LIN {X 0.171,Y -429.306,Z 1097.500,A 0.000,B 0.000,C 90.000,E1 269.943} C_DIS
LIN {X 0.033,Y -421.795,Z 1097.499,A 0.000,B 0.000,C 90.000,E1 269.771} C_DIS
LIN {X 0.153,Y -409.790,Z 1097.498,A 0.000,B 0.000,C 90.000,E1 269.542} C_DIS
LIN {X -0.190,Y -399.220,Z 1097.497,A 0.000,B 0.000,C 90.000,E1 269.484} C_DIS
LIN {X -0.102,Y -389.692,Z 1097.497,A 0.000,B 0.000,C 90.000,E1 269.427} C_DIS
LIN {X -0.076,Y -181.414,Z 1097.497,A 0.000,B 0.000,C 90.000,E1 269.427} C_DIS
LIN {X 0.018,Y -180.819,Z 1097.471,A 0.000,B 0.000,C 90.000,E1 264.837} C_DIS
LIN {X -0.083,Y -178.922,Z 1097.443,A 0.000,B 0.000,C 90.000,E1 259.803} C_DIS
LIN {X 0.003,Y -175.968,Z 1097.415,A 0.000,B 0.000,C 90.000,E1 254.685} C_DIS
LIN {X -0.050,Y -175.450,Z 1097.410,A 0.000,B 0.000,C 90.000,E1 253.850} C_DIS
LIN {X -0.041,Y -172.203,Z 1097.386,A 0.000,B 0.000,C 90.000,E1 249.571} C_DIS
LIN {X -0.062,Y -171.678,Z 1097.382,A 0.000,B 0.000,C 90.000,E1 248.720} C_DIS
LIN {X -0.072,Y -167.904,Z 1097.358,A 0.000,B 0.000,C 90.000,E1 244.409} C_DIS
LIN {X -0.053,Y -166.644,Z 1097.348,A 0.000,B 0.000,C 90.000,E1 242.666} C_DIS
LIN {X 0.002,Y -162.628,Z 1097.324,A 0.000,B 0.000,C 90.000,E1 238.280} C_DIS
LIN {X 0.061,Y -161.316,Z 1097.314,A 0.000,B 0.000,C 90.000,E1 236.501} C_DIS
LIN {X -0.029,Y -157.312,Z 1097.289,A 0.000,B 0.000,C 90.000,E1 232.110} C_DIS
LIN {X -0.097,Y -155.290,Z 1097.275,A 0.000,B 0.000,C 90.000,E1 229.461} C_DIS
LIN {X 0.050,Y -151.653,Z 1097.250,A 0.000,B 0.000,C 90.000,E1 224.919} C_DIS
LIN {X -0.013,Y -150.520,Z 1097.240,A 0.000,B 0.000,C 90.000,E1 223.137} C_DIS
LIN {X 0.011,Y -147.245,Z 1097.214,A 0.000,B 0.000,C 90.000,E1 218.588} C_DIS
LIN {X -0.025,Y -145.270,Z 1097.194,A 0.000,B 0.000,C 90.000,E1 214.945} C_DIS
LIN {X 0.009,Y -142.377,Z 1097.163,A 0.000,B 0.000,C 90.000,E1 209.411} C_DIS
LIN {X 0.059,Y -141.353,Z 1097.148,A 0.000,B 0.000,C 90.000,E1 206.616} C_DIS
LIN {X 0.042,Y -139.340,Z 1097.112,A 0.000,B 0.000,C 90.000,E1 200.120} C_DIS
LIN {X -0.039,Y -139.007,Z 1097.102,A 0.000,B 0.000,C 90.000,E1 198.290} C_DIS
LIN {X 0.048,Y -138.340,Z 1097.055,A 0.000,B 0.000,C 90.000,E1 189.849} C_DIS
LIN {X 0.071,Y -139.403,Z 1097.008,A 0.000,B 0.000,C 90.000,E1 181.432} C_DIS
LIN {X -0.015,Y -141.310,Z 1096.972,A 0.000,B 0.000,C 90.000,E1 174.951} C_DIS
LIN {X -0.058,Y -142.670,Z 1096.956,A 0.000,B 0.000,C 90.000,E1 172.186} C_DIS
LIN {X 0.064,Y -145.019,Z 1096.931,A 0.000,B 0.000,C 90.000,E1 167.521} C_DIS
LIN {X 0.021,Y -147.646,Z 1096.910,A 0.000,B 0.000,C 90.000,E1 163.866} C_DIS
LIN {X -0.043,Y -150.280,Z 1096.890,A 0.000,B 0.000,C 90.000,E1 160.242} C_DIS
LIN {X -0.030,Y -153.684,Z 1096.870,A 0.000,B 0.000,C 90.000,E1 156.613} C_DIS
LIN {X 0.025,Y -157.098,Z 1096.850,A 0.000,B 0.000,C 90.000,E1 152.999} C_DIS
LIN {X -0.037,Y -161.237,Z 1096.830,A 0.000,B 0.000,C 90.000,E1 149.459} C_DIS
LIN {X 0.048,Y -163.325,Z 1096.820,A 0.000,B 0.000,C 90.000,E1 147.661} C_DIS
LIN {X -0.081,Y -167.778,Z 1096.801,A 0.000,B 0.000,C 90.000,E1 144.196} C_DIS
LIN {X 0.071,Y -171.592,Z 1096.786,A 0.000,B 0.000,C 90.000,E1 141.537} C_DIS
LIN {X 0.002,Y -176.543,Z 1096.767,A 0.000,B 0.000,C 90.000,E1 138.119} C_DIS
LIN {X -0.006,Y -180.842,Z 1096.753,A 0.000,B 0.000,C 90.000,E1 135.567} C_DIS
LIN {X -0.022,Y -186.253,Z 1096.734,A 0.000,B 0.000,C 90.000,E1 132.204} C_DIS
LIN {X -0.084,Y -190.889,Z 1096.721,A 0.000,B 0.000,C 90.000,E1 129.725} C_DIS
LIN {X -0.051,Y -196.654,Z 1096.702,A 0.000,B 0.000,C 90.000,E1 126.423} C_DIS
LIN {X -0.056,Y -200.011,Z 1096.693,A 0.000,B 0.000,C 90.000,E1 124.739} C_DIS
LIN {X 0.114,Y -308.191,Z 1096.693,A 0.000,B 0.000,C 90.000,E1 124.692} C_DIS
LIN {X -0.031,Y -313.358,Z 1096.692,A 0.000,B 0.000,C 90.000,E1 124.532} C_DIS
LIN {X 0.081,Y -315.849,Z 1096.691,A 0.000,B 0.000,C 90.000,E1 124.326} C_DIS
LIN {X -0.136,Y -319.180,Z 1096.689,A 0.000,B 0.000,C 90.000,E1 123.992} C_DIS
LIN {X 0.031,Y -321.119,Z 1096.687,A 0.000,B 0.000,C 90.000,E1 123.658} C_DIS
LIN {X -0.070,Y -322.635,Z 1096.685,A 0.000,B 0.000,C 90.000,E1 123.372} C_DIS
LIN {X -0.076,Y -326.114,Z 1096.680,A 0.000,B 0.000,C 90.000,E1 122.418} C_DIS
LIN {X -0.078,Y -336.920,Z 1096.664,A 0.000,B 0.000,C 90.000,E1 119.589} C_DIS
LIN {X 0.023,Y -349.100,Z 1096.649,A 0.000,B 0.000,C 90.000,E1 116.796} C_DIS
LIN {X 0.009,Y -362.765,Z 1096.634,A 0.000,B 0.000,C 90.000,E1 114.079} C_DIS
LIN {X -0.006,Y -376.251,Z 1096.621,A 0.000,B 0.000,C 90.000,E1 111.716} C_DIS
LIN {X 0.043,Y -391.099,Z 1096.608,A 0.000,B 0.000,C 90.000,E1 109.396} C_DIS
LIN {X -0.045,Y -407.413,Z 1096.595,A 0.000,B 0.000,C 90.000,E1 107.149} C_DIS
LIN {X -0.100,Y -425.309,Z 1096.583,A 0.000,B 0.000,C 90.000,E1 104.954} C_DIS
LIN {X -0.142,Y -444.799,Z 1096.571,A 0.000,B 0.000,C 90.000,E1 102.827} C_DIS
LIN {X -0.016,Y -465.050,Z 1096.560,A 0.000,B 0.000,C 90.000,E1 100.838} C_DIS
LIN {X 0.001,Y -467.605,Z 1096.559,A 0.000,B 0.000,C 90.000,E1 100.602} C_DIS
LIN {X 0.018,Y -469.774,Z 1096.558,A 0.000,B 0.000,C 90.000,E1 100.366} C_DIS
LIN {X -0.217,Y -471.537,Z 1096.556,A 0.000,B 0.000,C 90.000,E1 100.141} C_DIS
LIN {X 0.098,Y -472.861,Z 1096.555,A 0.000,B 0.000,C 90.000,E1 99.849} C_DIS
LIN {X -0.186,Y -474.513,Z 1096.552,A 0.000,B 0.000,C 90.000,E1 99.378} C_DIS
LIN {X -0.072,Y -475.101,Z 1096.549,A 0.000,B 0.000,C 90.000,E1 98.859} C_DIS
LIN {X 0.056,Y -474.725,Z 1096.546,A 0.000,B 0.000,C 90.000,E1 98.341} C_DIS
LIN {X 0.253,Y -473.330,Z 1096.544,A 0.000,B 0.000,C 90.000,E1 97.814} C_DIS
LIN {X 0.050,Y -472.179,Z 1096.542,A 0.000,B 0.000,C 90.000,E1 97.587} C_DIS
LIN {X -0.088,Y -470.646,Z 1096.541,A 0.000,B 0.000,C 90.000,E1 97.352} C_DIS
LIN {X -0.214,Y -456.164,Z 1096.530,A 0.000,B 0.000,C 90.000,E1 95.334} C_DIS
LIN {X -0.079,Y -440.261,Z 1096.516,A 0.000,B 0.000,C 90.000,E1 92.980} C_DIS
LIN {X 0.048,Y -425.629,Z 1096.503,A 0.000,B 0.000,C 90.000,E1 90.573} C_DIS
LIN {X 0.049,Y -407.500,Z 1096.485,A 0.000,B 0.000,C 90.000,E1 87.306} C_DIS
LIN {X 0.079,Y -397.005,Z 1096.474,A 0.000,B 0.000,C 90.000,E1 85.355} C_DIS
LIN {X -0.034,Y -386.300,Z 1096.463,A 0.000,B 0.000,C 90.000,E1 83.394} C_DIS
LIN {X 0.053,Y -377.169,Z 1096.454,A 0.000,B 0.000,C 90.000,E1 81.659} C_DIS
LIN {X -0.034,Y -367.668,Z 1096.444,A 0.000,B 0.000,C 90.000,E1 79.926} C_DIS
LIN {X -0.166,Y -357.876,Z 1096.434,A 0.000,B 0.000,C 90.000,E1 78.173} C_DIS
LIN {X -0.039,Y -346.268,Z 1096.422,A 0.000,B 0.000,C 90.000,E1 76.047} C_DIS
LIN {X 0.148,Y -333.118,Z 1096.409,A 0.000,B 0.000,C 90.000,E1 73.559} C_DIS
LIN {X 0.013,Y -315.862,Z 1096.390,A 0.000,B 0.000,C 90.000,E1 70.115} C_DIS
LIN {X -0.145,Y -302.718,Z 1096.373,A 0.000,B 0.000,C 90.000,E1 67.230} C_DIS
LIN {X -0.035,Y -292.864,Z 1096.360,A 0.000,B 0.000,C 90.000,E1 64.897} C_DIS
LIN {X -0.178,Y -281.874,Z 1096.346,A 0.000,B 0.000,C 90.000,E1 62.231} C_DIS
LIN {X -0.070,Y -271.125,Z 1096.330,A 0.000,B 0.000,C 90.000,E1 59.459} C_DIS
LIN {X -0.053,Y -259.422,Z 1096.313,A 0.000,B 0.000,C 90.000,E1 56.294} C_DIS
LIN {X 0.000,Y -248.215,Z 1096.295,A 0.000,B 0.000,C 90.000,E1 53.050} C_DIS
LIN {X -0.007,Y -237.844,Z 1096.276,A 0.000,B 0.000,C 90.000,E1 49.747} C_DIS
LIN {X -0.005,Y -228.242,Z 1096.258,A 0.000,B 0.000,C 90.000,E1 46.377} C_DIS
LIN {X -0.035,Y -220.174,Z 1096.241,A 0.000,B 0.000,C 90.000,E1 43.338} C_DIS
LIN {X -0.086,Y -212.478,Z 1096.224,A 0.000,B 0.000,C 90.000,E1 40.253} C_DIS
LIN {X 0.013,Y -205.151,Z 1096.206,A 0.000,B 0.000,C 90.000,E1 37.076} C_DIS
LIN {X 0.052,Y -198.373,Z 1096.188,A 0.000,B 0.000,C 90.000,E1 33.865} C_DIS
LIN {X -0.122,Y -192.214,Z 1096.170,A 0.000,B 0.000,C 90.000,E1 30.669} C_DIS
LIN {X 0.023,Y -186.724,Z 1096.152,A 0.000,B 0.000,C 90.000,E1 27.334} C_DIS
LIN {X -0.055,Y -181.962,Z 1096.133,A 0.000,B 0.000,C 90.000,E1 24.027} C_DIS
LIN {X -0.053,Y -176.995,Z 1096.110,A 0.000,B 0.000,C 90.000,E1 19.812} C_DIS
LIN {X -0.055,Y -173.062,Z 1096.086,A 0.000,B 0.000,C 90.000,E1 15.552} C_DIS
LIN {X 0.016,Y -169.745,Z 1096.058,A 0.000,B 0.000,C 90.000,E1 10.366} C_DIS
LIN {X -0.011,Y -167.547,Z 1096.019,A 0.000,B 0.000,C 90.000,E1 3.440} C_DIS
LIN {X -0.017,Y -168.706,Z 1095.964,A 0.000,B 0.000,C 90.000,E1 353.451} C_DIS
LIN {X 0.055,Y -171.259,Z 1095.935,A 0.000,B 0.000,C 90.000,E1 348.229} C_DIS
LIN {X 0.070,Y -174.548,Z 1095.911,A 0.000,B 0.000,C 90.000,E1 343.921} C_DIS
LIN {X -0.075,Y -178.893,Z 1095.887,A 0.000,B 0.000,C 90.000,E1 339.699} C_DIS
LIN {X -0.044,Y -183.100,Z 1095.868,A 0.000,B 0.000,C 90.000,E1 336.305} C_DIS
LIN {X -0.023,Y -188.059,Z 1095.850,A 0.000,B 0.000,C 90.000,E1 332.948} C_DIS
LIN {X 0.046,Y -193.760,Z 1095.831,A 0.000,B 0.000,C 90.000,E1 329.616} C_DIS
LIN {X -0.047,Y -200.207,Z 1095.813,A 0.000,B 0.000,C 90.000,E1 326.373} C_DIS
LIN {X 0.027,Y -207.316,Z 1095.795,A 0.000,B 0.000,C 90.000,E1 323.130} C_DIS
LIN {X -0.076,Y -215.345,Z 1095.778,A 0.000,B 0.000,C 90.000,E1 319.989} C_DIS
LIN {X -0.018,Y -224.059,Z 1095.760,A 0.000,B 0.000,C 90.000,E1 316.863} C_DIS
LIN {X 0.089,Y -233.756,Z 1095.743,A 0.000,B 0.000,C 90.000,E1 313.785} C_DIS
LIN {X -0.018,Y -243.414,Z 1095.729,A 0.000,B 0.000,C 90.000,E1 311.191} C_DIS
LIN {X -0.037,Y -252.645,Z 1095.717,A 0.000,B 0.000,C 90.000,E1 308.991} C_DIS
LIN {X 0.077,Y -266.395,Z 1095.701,A 0.000,B 0.000,C 90.000,E1 306.091} C_DIS
LIN {X 0.080,Y -281.412,Z 1095.685,A 0.000,B 0.000,C 90.000,E1 303.293} C_DIS
LIN {X -0.005,Y -299.593,Z 1095.668,A 0.000,B 0.000,C 90.000,E1 300.256} C_DIS
LIN {X -0.016,Y -319.577,Z 1095.652,A 0.000,B 0.000,C 90.000,E1 297.308} C_DIS
LIN {X 0.009,Y -336.467,Z 1095.639,A 0.000,B 0.000,C 90.000,E1 295.079} C_DIS
LIN {X -0.080,Y -349.541,Z 1095.631,A 0.000,B 0.000,C 90.000,E1 293.567} C_DIS
LIN {X -0.194,Y -362.823,Z 1095.623,A 0.000,B 0.000,C 90.000,E1 292.153} C_DIS
LIN {X -0.066,Y -376.176,Z 1095.616,A 0.000,B 0.000,C 90.000,E1 290.844} C_DIS
LIN {X -0.076,Y -395.554,Z 1095.606,A 0.000,B 0.000,C 90.000,E1 289.141} C_DIS
LIN {X 0.030,Y -409.102,Z 1095.600,A 0.000,B 0.000,C 90.000,E1 287.946} C_DIS
LIN {X 0.036,Y -419.690,Z 1095.594,A 0.000,B 0.000,C 90.000,E1 286.985} C_DIS
LIN {X -0.079,Y -427.432,Z 1095.590,A 0.000,B 0.000,C 90.000,E1 286.260} C_DIS
LIN {X 0.023,Y -434.966,Z 1095.586,A 0.000,B 0.000,C 90.000,E1 285.481} C_DIS
LIN {X -0.185,Y -442.194,Z 1095.582,A 0.000,B 0.000,C 90.000,E1 284.717} C_DIS
LIN {X 0.151,Y -448.956,Z 1095.577,A 0.000,B 0.000,C 90.000,E1 283.883} C_DIS
LIN {X -0.002,Y -455.110,Z 1095.573,A 0.000,B 0.000,C 90.000,E1 283.119} C_DIS
LIN {X 0.075,Y -458.896,Z 1095.570,A 0.000,B 0.000,C 90.000,E1 282.591} C_DIS
LIN {X 0.013,Y -463.916,Z 1095.566,A 0.000,B 0.000,C 90.000,E1 281.827} C_DIS
LIN {X -0.104,Y -468.213,Z 1095.561,A 0.000,B 0.000,C 90.000,E1 281.074} C_DIS
LIN {X -0.089,Y -471.792,Z 1095.557,A 0.000,B 0.000,C 90.000,E1 280.310} C_DIS
LIN {X -0.130,Y -474.745,Z 1095.553,A 0.000,B 0.000,C 90.000,E1 279.557} C_DIS
LIN {X 0.060,Y -476.344,Z 1095.550,A 0.000,B 0.000,C 90.000,E1 279.029} C_DIS
LIN {X 0.187,Y -477.748,Z 1095.547,A 0.000,B 0.000,C 90.000,E1 278.511} C_DIS
LIN {X -0.147,Y -478.896,Z 1095.545,A 0.000,B 0.000,C 90.000,E1 278.049} C_DIS
LIN {X 0.002,Y -479.796,Z 1095.542,A 0.000,B 0.000,C 90.000,E1 277.530} C_DIS
LIN {X 0.159,Y -480.516,Z 1095.539,A 0.000,B 0.000,C 90.000,E1 277.011} C_DIS
LIN {X -0.100,Y -480.986,Z 1095.536,A 0.000,B 0.000,C 90.000,E1 276.543} C_DIS
LIN {X 0.013,Y -481.163,Z 1095.534,A 0.000,B 0.000,C 90.000,E1 276.030} C_DIS
LIN {X 0.183,Y -480.992,Z 1095.531,A 0.000,B 0.000,C 90.000,E1 275.511} C_DIS
LIN {X -0.127,Y -480.502,Z 1095.528,A 0.000,B 0.000,C 90.000,E1 275.049} C_DIS
LIN {X 0.040,Y -479.609,Z 1095.525,A 0.000,B 0.000,C 90.000,E1 274.531} C_DIS
LIN {X 0.200,Y -478.204,Z 1095.522,A 0.000,B 0.000,C 90.000,E1 274.012} C_DIS
LIN {X -0.153,Y -476.301,Z 1095.520,A 0.000,B 0.000,C 90.000,E1 273.555} C_DIS
LIN {X -0.009,Y -473.740,Z 1095.517,A 0.000,B 0.000,C 90.000,E1 273.037} C_DIS
LIN {X 0.092,Y -470.356,Z 1095.514,A 0.000,B 0.000,C 90.000,E1 272.522} C_DIS
LIN {X 0.176,Y -466.075,Z 1095.511,A 0.000,B 0.000,C 90.000,E1 272.007} C_DIS
LIN {X -0.209,Y -460.563,Z 1095.508,A 0.000,B 0.000,C 90.000,E1 271.547} C_DIS
LIN {X -0.209,Y -457.683,Z 1095.507,A 0.000,B 0.000,C 90.000,E1 271.318} C_DIS
LIN {X 0.070,Y -451.340,Z 1095.505,A 0.000,B 0.000,C 90.000,E1 270.859} C_DIS
LIN {X -0.058,Y -444.673,Z 1095.503,A 0.000,B 0.000,C 90.000,E1 270.516} C_DIS
LIN {X -0.168,Y -437.586,Z 1095.501,A 0.000,B 0.000,C 90.000,E1 270.229} C_DIS
LIN {X 0.135,Y -430.141,Z 1095.500,A 0.000,B 0.000,C 90.000,E1 269.943} C_DIS
LIN {X -0.039,Y -422.384,Z 1095.499,A 0.000,B 0.000,C 90.000,E1 269.771} C_DIS
LIN {X 0.123,Y -414.688,Z 1095.498,A 0.000,B 0.000,C 90.000,E1 269.599} C_DIS
LIN {X 0.116,Y -406.084,Z 1095.497,A 0.000,B 0.000,C 90.000,E1 269.484} C_DIS
LIN {X -0.095,Y -394.535,Z 1095.497,A 0.000,B 0.000,C 90.000,E1 269.427} C_DIS
LIN {X -0.159,Y -391.661,Z 1095.497,A 0.000,B 0.000,C 90.000,E1 269.427} C_DIS
LIN {X 0.078,Y -181.412,Z 1095.497,A 0.000,B 0.000,C 90.000,E1 269.370} C_DIS
LIN {X -0.012,Y -180.816,Z 1095.471,A 0.000,B 0.000,C 90.000,E1 264.837} C_DIS
LIN {X 0.066,Y -178.919,Z 1095.443,A 0.000,B 0.000,C 90.000,E1 259.746} C_DIS
LIN {X -0.025,Y -175.964,Z 1095.415,A 0.000,B 0.000,C 90.000,E1 254.685} C_DIS
LIN {X 0.090,Y -175.441,Z 1095.410,A 0.000,B 0.000,C 90.000,E1 253.795} C_DIS
LIN {X -0.068,Y -172.198,Z 1095.386,A 0.000,B 0.000,C 90.000,E1 249.571} C_DIS
LIN {X -0.091,Y -171.671,Z 1095.382,A 0.000,B 0.000,C 90.000,E1 248.720} C_DIS
LIN {X -0.099,Y -167.897,Z 1095.358,A 0.000,B 0.000,C 90.000,E1 244.409} C_DIS
LIN {X 0.068,Y -166.636,Z 1095.348,A 0.000,B 0.000,C 90.000,E1 242.615} C_DIS
LIN {X -0.025,Y -162.622,Z 1095.324,A 0.000,B 0.000,C 90.000,E1 238.280} C_DIS
LIN {X 0.034,Y -161.308,Z 1095.314,A 0.000,B 0.000,C 90.000,E1 236.501} C_DIS
LIN {X -0.056,Y -157.305,Z 1095.289,A 0.000,B 0.000,C 90.000,E1 232.110} C_DIS
LIN {X 0.096,Y -155.281,Z 1095.275,A 0.000,B 0.000,C 90.000,E1 229.380} C_DIS
LIN {X 0.024,Y -151.646,Z 1095.250,A 0.000,B 0.000,C 90.000,E1 224.919} C_DIS
LIN {X -0.039,Y -150.515,Z 1095.240,A 0.000,B 0.000,C 90.000,E1 223.137} C_DIS
LIN {X -0.015,Y -147.239,Z 1095.214,A 0.000,B 0.000,C 90.000,E1 218.588} C_DIS
LIN {X -0.050,Y -145.263,Z 1095.194,A 0.000,B 0.000,C 90.000,E1 214.945} C_DIS
LIN {X -0.016,Y -142.373,Z 1095.163,A 0.000,B 0.000,C 90.000,E1 209.411} C_DIS
LIN {X -0.020,Y -141.758,Z 1095.153,A 0.000,B 0.000,C 90.000,E1 207.564} C_DIS
LIN {X 0.030,Y -139.498,Z 1095.117,A 0.000,B 0.000,C 90.000,E1 201.046} C_DIS
LIN {X 0.067,Y -139.004,Z 1095.101,A 0.000,B 0.000,C 90.000,E1 198.236} C_DIS
LIN {X 0.024,Y -138.339,Z 1095.055,A 0.000,B 0.000,C 90.000,E1 189.849} C_DIS
LIN {X 0.046,Y -139.406,Z 1095.008,A 0.000,B 0.000,C 90.000,E1 181.432} C_DIS
LIN {X -0.040,Y -141.314,Z 1094.972,A 0.000,B 0.000,C 90.000,E1 174.951} C_DIS
LIN {X 0.057,Y -142.673,Z 1094.956,A 0.000,B 0.000,C 90.000,E1 172.129} C_DIS
LIN {X 0.039,Y -145.026,Z 1094.931,A 0.000,B 0.000,C 90.000,E1 167.521} C_DIS
LIN {X -0.005,Y -147.652,Z 1094.910,A 0.000,B 0.000,C 90.000,E1 163.866} C_DIS
LIN {X -0.070,Y -150.288,Z 1094.890,A 0.000,B 0.000,C 90.000,E1 160.242} C_DIS
LIN {X -0.057,Y -153.695,Z 1094.870,A 0.000,B 0.000,C 90.000,E1 156.613} C_DIS
LIN {X -0.002,Y -157.108,Z 1094.850,A 0.000,B 0.000,C 90.000,E1 152.999} C_DIS
LIN {X -0.065,Y -161.250,Z 1094.830,A 0.000,B 0.000,C 90.000,E1 149.459} C_DIS
LIN {X 0.021,Y -163.336,Z 1094.820,A 0.000,B 0.000,C 90.000,E1 147.661} C_DIS
LIN {X 0.027,Y -167.791,Z 1094.801,A 0.000,B 0.000,C 90.000,E1 144.149} C_DIS
LIN {X 0.043,Y -171.605,Z 1094.786,A 0.000,B 0.000,C 90.000,E1 141.537} C_DIS
LIN {X 0.091,Y -176.559,Z 1094.767,A 0.000,B 0.000,C 90.000,E1 138.081} C_DIS
LIN {X -0.036,Y -180.857,Z 1094.753,A 0.000,B 0.000,C 90.000,E1 135.567} C_DIS
LIN {X -0.051,Y -186.269,Z 1094.734,A 0.000,B 0.000,C 90.000,E1 132.204} C_DIS
LIN {X 0.008,Y -190.905,Z 1094.720,A 0.000,B 0.000,C 90.000,E1 129.688} C_DIS
LIN {X 0.076,Y -196.671,Z 1094.702,A 0.000,B 0.000,C 90.000,E1 126.377} C_DIS
LIN {X 0.062,Y -199.941,Z 1094.693,A 0.000,B 0.000,C 90.000,E1 124.739} C_DIS
LIN {X 0.059,Y -307.476,Z 1094.693,A 0.000,B 0.000,C 90.000,E1 124.739} C_DIS
LIN {X 0.066,Y -309.988,Z 1094.693,A 0.000,B 0.000,C 90.000,E1 124.692} C_DIS
LIN {X -0.080,Y -313.832,Z 1094.692,A 0.000,B 0.000,C 90.000,E1 124.532} C_DIS
LIN {X 0.032,Y -316.142,Z 1094.691,A 0.000,B 0.000,C 90.000,E1 124.326} C_DIS
LIN {X -0.185,Y -319.328,Z 1094.689,A 0.000,B 0.000,C 90.000,E1 123.992} C_DIS
LIN {X -0.074,Y -321.258,Z 1094.687,A 0.000,B 0.000,C 90.000,E1 123.658} C_DIS
LIN {X 0.217,Y -322.762,Z 1094.685,A 0.000,B 0.000,C 90.000,E1 123.293} C_DIS
LIN {X 0.051,Y -337.012,Z 1094.664,A 0.000,B 0.000,C 90.000,E1 119.539} C_DIS
LIN {X 0.168,Y -349.206,Z 1094.649,A 0.000,B 0.000,C 90.000,E1 116.744} C_DIS
LIN {X -0.161,Y -362.886,Z 1094.634,A 0.000,B 0.000,C 90.000,E1 114.079} C_DIS
LIN {X -0.180,Y -376.387,Z 1094.620,A 0.000,B 0.000,C 90.000,E1 111.716} C_DIS
LIN {X -0.134,Y -391.250,Z 1094.608,A 0.000,B 0.000,C 90.000,E1 109.396} C_DIS
LIN {X 0.164,Y -407.581,Z 1094.595,A 0.000,B 0.000,C 90.000,E1 107.094} C_DIS
LIN {X 0.127,Y -425.496,Z 1094.583,A 0.000,B 0.000,C 90.000,E1 104.898} C_DIS
LIN {X 0.109,Y -444.998,Z 1094.571,A 0.000,B 0.000,C 90.000,E1 102.771} C_DIS
LIN {X -0.192,Y -465.257,Z 1094.560,A 0.000,B 0.000,C 90.000,E1 100.838} C_DIS
LIN {X -0.174,Y -467.803,Z 1094.559,A 0.000,B 0.000,C 90.000,E1 100.602} C_DIS
LIN {X -0.157,Y -469.911,Z 1094.557,A 0.000,B 0.000,C 90.000,E1 100.366} C_DIS
LIN {X 0.155,Y -471.631,Z 1094.556,A 0.000,B 0.000,C 90.000,E1 100.074} C_DIS
LIN {X -0.077,Y -472.922,Z 1094.555,A 0.000,B 0.000,C 90.000,E1 99.849} C_DIS
LIN {X 0.107,Y -474.525,Z 1094.552,A 0.000,B 0.000,C 90.000,E1 99.321} C_DIS
LIN {X 0.224,Y -475.071,Z 1094.549,A 0.000,B 0.000,C 90.000,E1 98.803} C_DIS
LIN {X -0.118,Y -474.653,Z 1094.546,A 0.000,B 0.000,C 90.000,E1 98.341} C_DIS
LIN {X 0.079,Y -473.211,Z 1094.543,A 0.000,B 0.000,C 90.000,E1 97.814} C_DIS
LIN {X -0.123,Y -472.031,Z 1094.542,A 0.000,B 0.000,C 90.000,E1 97.587} C_DIS
LIN {X 0.206,Y -470.462,Z 1094.541,A 0.000,B 0.000,C 90.000,E1 97.296} C_DIS
LIN {X 0.069,Y -456.006,Z 1094.529,A 0.000,B 0.000,C 90.000,E1 95.277} C_DIS
LIN {X 0.191,Y -440.105,Z 1094.516,A 0.000,B 0.000,C 90.000,E1 92.922} C_DIS
LIN {X -0.121,Y -425.471,Z 1094.503,A 0.000,B 0.000,C 90.000,E1 90.573} C_DIS
LIN {X -0.118,Y -407.373,Z 1094.485,A 0.000,B 0.000,C 90.000,E1 87.306} C_DIS
LIN {X -0.086,Y -396.877,Z 1094.474,A 0.000,B 0.000,C 90.000,E1 85.355} C_DIS
LIN {X 0.187,Y -386.154,Z 1094.463,A 0.000,B 0.000,C 90.000,E1 83.337} C_DIS
LIN {X -0.108,Y -377.019,Z 1094.454,A 0.000,B 0.000,C 90.000,E1 81.659} C_DIS
LIN {X -0.129,Y -367.483,Z 1094.444,A 0.000,B 0.000,C 90.000,E1 79.916} C_DIS
LIN {X 0.024,Y -357.661,Z 1094.434,A 0.000,B 0.000,C 90.000,E1 78.117} C_DIS
LIN {X 0.138,Y -346.059,Z 1094.422,A 0.000,B 0.000,C 90.000,E1 75.992} C_DIS
LIN {X -0.124,Y -331.289,Z 1094.407,A 0.000,B 0.000,C 90.000,E1 73.268} C_DIS
LIN {X 0.153,Y -315.668,Z 1094.389,A 0.000,B 0.000,C 90.000,E1 70.061} C_DIS
LIN {X -0.021,Y -302.546,Z 1094.373,A 0.000,B 0.000,C 90.000,E1 67.177} C_DIS
LIN {X 0.077,Y -292.684,Z 1094.360,A 0.000,B 0.000,C 90.000,E1 64.845} C_DIS
LIN {X 0.051,Y -281.675,Z 1094.345,A 0.000,B 0.000,C 90.000,E1 62.153} C_DIS
LIN {X 0.012,Y -270.918,Z 1094.330,A 0.000,B 0.000,C 90.000,E1 59.410} C_DIS
LIN {X -0.105,Y -260.470,Z 1094.314,A 0.000,B 0.000,C 90.000,E1 56.628} C_DIS
LIN {X -0.040,Y -250.420,Z 1094.299,A 0.000,B 0.000,C 90.000,E1 53.749} C_DIS
LIN {X 0.055,Y -239.828,Z 1094.280,A 0.000,B 0.000,C 90.000,E1 50.436} C_DIS
LIN {X 0.100,Y -230.051,Z 1094.262,A 0.000,B 0.000,C 90.000,E1 47.067} C_DIS
LIN {X 0.111,Y -221.895,Z 1094.245,A 0.000,B 0.000,C 90.000,E1 44.028} C_DIS
LIN {X -0.068,Y -214.054,Z 1094.228,A 0.000,B 0.000,C 90.000,E1 40.987} C_DIS
LIN {X 0.070,Y -206.616,Z 1094.210,A 0.000,B 0.000,C 90.000,E1 37.810} C_DIS
LIN {X 0.095,Y -199.664,Z 1094.192,A 0.000,B 0.000,C 90.000,E1 34.612} C_DIS
LIN {X 0.051,Y -193.336,Z 1094.174,A 0.000,B 0.000,C 90.000,E1 31.386} C_DIS
LIN {X 0.049,Y -187.706,Z 1094.156,A 0.000,B 0.000,C 90.000,E1 28.103} C_DIS
LIN {X 0.070,Y -182.784,Z 1094.138,A 0.000,B 0.000,C 90.000,E1 24.771} C_DIS
LIN {X 0.074,Y -178.580,Z 1094.119,A 0.000,B 0.000,C 90.000,E1 21.408} C_DIS
LIN {X 0.058,Y -174.217,Z 1094.095,A 0.000,B 0.000,C 90.000,E1 17.166} C_DIS
LIN {X 0.044,Y -170.975,Z 1094.072,A 0.000,B 0.000,C 90.000,E1 12.883} C_DIS
LIN {X 0.035,Y -168.371,Z 1094.043,A 0.000,B 0.000,C 90.000,E1 7.701} C_DIS
LIN {X -0.056,Y -169.131,Z 1093.954,A 0.000,B 0.000,C 90.000,E1 351.724} C_DIS
LIN {X -0.015,Y -172.198,Z 1093.925,A 0.000,B 0.000,C 90.000,E1 346.520} C_DIS
LIN {X -0.045,Y -175.946,Z 1093.901,A 0.000,B 0.000,C 90.000,E1 342.236} C_DIS
LIN {X -0.039,Y -179.662,Z 1093.882,A 0.000,B 0.000,C 90.000,E1 338.827} C_DIS
LIN {X 0.013,Y -184.054,Z 1093.864,A 0.000,B 0.000,C 90.000,E1 335.433} C_DIS
LIN {X -0.029,Y -189.201,Z 1093.845,A 0.000,B 0.000,C 90.000,E1 332.103} C_DIS
LIN {X 0.000,Y -195.124,Z 1093.827,A 0.000,B 0.000,C 90.000,E1 328.791} C_DIS
LIN {X 0.057,Y -201.693,Z 1093.808,A 0.000,B 0.000,C 90.000,E1 325.515} C_DIS
LIN {X 0.013,Y -209.099,Z 1093.791,A 0.000,B 0.000,C 90.000,E1 322.316} C_DIS
LIN {X 0.018,Y -218.349,Z 1093.771,A 0.000,B 0.000,C 90.000,E1 318.771} C_DIS
LIN {X -0.011,Y -227.406,Z 1093.754,A 0.000,B 0.000,C 90.000,E1 315.688} C_DIS
LIN {X 0.066,Y -236.239,Z 1093.739,A 0.000,B 0.000,C 90.000,E1 313.014} C_DIS
LIN {X 0.041,Y -246.256,Z 1093.725,A 0.000,B 0.000,C 90.000,E1 310.415} C_DIS
LIN {X 0.050,Y -255.841,Z 1093.712,A 0.000,B 0.000,C 90.000,E1 308.222} C_DIS
LIN {X -0.072,Y -269.957,Z 1093.697,A 0.000,B 0.000,C 90.000,E1 305.391} C_DIS
LIN {X -0.140,Y -285.314,Z 1093.681,A 0.000,B 0.000,C 90.000,E1 302.625} C_DIS
LIN {X 0.142,Y -303.898,Z 1093.664,A 0.000,B 0.000,C 90.000,E1 299.539} C_DIS
LIN {X 0.124,Y -324.303,Z 1093.648,A 0.000,B 0.000,C 90.000,E1 296.616} C_DIS
LIN {X -0.159,Y -339.087,Z 1093.637,A 0.000,B 0.000,C 90.000,E1 294.771} C_DIS
LIN {X 0.076,Y -360.518,Z 1093.624,A 0.000,B 0.000,C 90.000,E1 292.333} C_DIS
LIN {X -0.095,Y -373.945,Z 1093.617,A 0.000,B 0.000,C 90.000,E1 291.046} C_DIS
LIN {X 0.129,Y -395.786,Z 1093.606,A 0.000,B 0.000,C 90.000,E1 289.087} C_DIS
LIN {X -0.193,Y -409.399,Z 1093.599,A 0.000,B 0.000,C 90.000,E1 287.946} C_DIS
LIN {X -0.144,Y -417.381,Z 1093.596,A 0.000,B 0.000,C 90.000,E1 287.221} C_DIS
LIN {X 0.183,Y -425.193,Z 1093.591,A 0.000,B 0.000,C 90.000,E1 286.441} C_DIS
LIN {X 0.003,Y -432.714,Z 1093.587,A 0.000,B 0.000,C 90.000,E1 285.717} C_DIS
LIN {X -0.173,Y -440.085,Z 1093.583,A 0.000,B 0.000,C 90.000,E1 284.954} C_DIS
LIN {X 0.145,Y -447.039,Z 1093.578,A 0.000,B 0.000,C 90.000,E1 284.120} C_DIS
LIN {X -0.020,Y -453.381,Z 1093.574,A 0.000,B 0.000,C 90.000,E1 283.355} C_DIS
LIN {X -0.136,Y -459.152,Z 1093.570,A 0.000,B 0.000,C 90.000,E1 282.591} C_DIS
LIN {X -0.198,Y -464.157,Z 1093.566,A 0.000,B 0.000,C 90.000,E1 281.827} C_DIS
LIN {X -0.066,Y -467.109,Z 1093.563,A 0.000,B 0.000,C 90.000,E1 281.299} C_DIS
LIN {X -0.154,Y -470.891,Z 1093.558,A 0.000,B 0.000,C 90.000,E1 280.546} C_DIS
LIN {X 0.020,Y -473.072,Z 1093.556,A 0.000,B 0.000,C 90.000,E1 280.018} C_DIS
LIN {X 0.128,Y -474.972,Z 1093.553,A 0.000,B 0.000,C 90.000,E1 279.500} C_DIS
LIN {X -0.149,Y -476.549,Z 1093.550,A 0.000,B 0.000,C 90.000,E1 279.029} C_DIS
LIN {X -0.022,Y -477.923,Z 1093.547,A 0.000,B 0.000,C 90.000,E1 278.511} C_DIS
LIN {X 0.119,Y -479.055,Z 1093.544,A 0.000,B 0.000,C 90.000,E1 277.992} C_DIS
LIN {X -0.206,Y -480.000,Z 1093.542,A 0.000,B 0.000,C 90.000,E1 277.530} C_DIS
LIN {X 0.011,Y -480.733,Z 1093.539,A 0.000,B 0.000,C 90.000,E1 277.004} C_DIS
LIN {X 0.171,Y -481.182,Z 1093.536,A 0.000,B 0.000,C 90.000,E1 276.486} C_DIS
LIN {X -0.141,Y -481.381,Z 1093.533,A 0.000,B 0.000,C 90.000,E1 276.024} C_DIS
LIN {X -0.021,Y -481.254,Z 1093.531,A 0.000,B 0.000,C 90.000,E1 275.511} C_DIS
LIN {X 0.151,Y -480.758,Z 1093.528,A 0.000,B 0.000,C 90.000,E1 274.992} C_DIS
LIN {X -0.160,Y -479.832,Z 1093.525,A 0.000,B 0.000,C 90.000,E1 274.531} C_DIS
LIN {X 0.002,Y -478.483,Z 1093.522,A 0.000,B 0.000,C 90.000,E1 274.012} C_DIS
LIN {X 0.127,Y -476.549,Z 1093.520,A 0.000,B 0.000,C 90.000,E1 273.498} C_DIS
LIN {X -0.202,Y -473.979,Z 1093.517,A 0.000,B 0.000,C 90.000,E1 273.037} C_DIS
LIN {X -0.099,Y -470.584,Z 1093.514,A 0.000,B 0.000,C 90.000,E1 272.522} C_DIS
LIN {X -0.012,Y -466.238,Z 1093.511,A 0.000,B 0.000,C 90.000,E1 272.007} C_DIS
LIN {X 0.067,Y -460.767,Z 1093.508,A 0.000,B 0.000,C 90.000,E1 271.489} C_DIS
LIN {X 0.021,Y -454.507,Z 1093.506,A 0.000,B 0.000,C 90.000,E1 271.031} C_DIS
LIN {X 0.058,Y -447.822,Z 1093.504,A 0.000,B 0.000,C 90.000,E1 270.630} C_DIS
LIN {X 0.159,Y -440.898,Z 1093.502,A 0.000,B 0.000,C 90.000,E1 270.286} C_DIS
LIN {X -0.153,Y -433.585,Z 1093.500,A 0.000,B 0.000,C 90.000,E1 270.057} C_DIS
LIN {X -0.034,Y -425.904,Z 1093.499,A 0.000,B 0.000,C 90.000,E1 269.828} C_DIS
LIN {X 0.035,Y -418.330,Z 1093.498,A 0.000,B 0.000,C 90.000,E1 269.656} C_DIS
LIN {X -0.080,Y -410.064,Z 1093.497,A 0.000,B 0.000,C 90.000,E1 269.542} C_DIS
LIN {X -0.086,Y -397.424,Z 1093.497,A 0.000,B 0.000,C 90.000,E1 269.427} C_DIS
LIN {X 0.120,Y -390.627,Z 1093.497,A 0.000,B 0.000,C 90.000,E1 269.370} C_DIS
LIN {X 0.027,Y -181.408,Z 1093.497,A 0.000,B 0.000,C 90.000,E1 269.370} C_DIS
LIN {X -0.061,Y -180.810,Z 1093.471,A 0.000,B 0.000,C 90.000,E1 264.837} C_DIS
LIN {X 0.016,Y -178.913,Z 1093.443,A 0.000,B 0.000,C 90.000,E1 259.746} C_DIS
LIN {X 0.095,Y -175.957,Z 1093.415,A 0.000,B 0.000,C 90.000,E1 254.629} C_DIS
LIN {X 0.042,Y -175.428,Z 1093.410,A 0.000,B 0.000,C 90.000,E1 253.795} C_DIS
LIN {X 0.045,Y -172.188,Z 1093.386,A 0.000,B 0.000,C 90.000,E1 249.518} C_DIS
LIN {X 0.021,Y -171.660,Z 1093.381,A 0.000,B 0.000,C 90.000,E1 248.666} C_DIS
LIN {X 0.005,Y -167.884,Z 1093.358,A 0.000,B 0.000,C 90.000,E1 244.357} C_DIS
LIN {X 0.020,Y -166.621,Z 1093.348,A 0.000,B 0.000,C 90.000,E1 242.615} C_DIS
LIN {X 0.014,Y -162.608,Z 1093.324,A 0.000,B 0.000,C 90.000,E1 238.250} C_DIS
LIN {X -0.013,Y -161.293,Z 1093.314,A 0.000,B 0.000,C 90.000,E1 236.501} C_DIS
LIN {X 0.022,Y -157.291,Z 1093.289,A 0.000,B 0.000,C 90.000,E1 232.065} C_DIS
LIN {X 0.045,Y -156.008,Z 1093.279,A 0.000,B 0.000,C 90.000,E1 230.275} C_DIS
LIN {X 0.005,Y -152.267,Z 1093.255,A 0.000,B 0.000,C 90.000,E1 225.810} C_DIS
LIN {X 0.027,Y -150.504,Z 1093.240,A 0.000,B 0.000,C 90.000,E1 223.095} C_DIS
LIN {X 0.056,Y -147.229,Z 1093.214,A 0.000,B 0.000,C 90.000,E1 218.543} C_DIS
LIN {X 0.026,Y -145.251,Z 1093.194,A 0.000,B 0.000,C 90.000,E1 214.898} C_DIS
LIN {X -0.058,Y -142.366,Z 1093.163,A 0.000,B 0.000,C 90.000,E1 209.411} C_DIS
LIN {X 0.062,Y -141.752,Z 1093.153,A 0.000,B 0.000,C 90.000,E1 207.513} C_DIS
LIN {X -0.011,Y -139.495,Z 1093.117,A 0.000,B 0.000,C 90.000,E1 201.046} C_DIS
LIN {X 0.026,Y -139.000,Z 1093.101,A 0.000,B 0.000,C 90.000,E1 198.236} C_DIS
LIN {X -0.018,Y -138.338,Z 1093.055,A 0.000,B 0.000,C 90.000,E1 189.849} C_DIS
LIN {X 0.004,Y -139.411,Z 1093.008,A 0.000,B 0.000,C 90.000,E1 181.432} C_DIS
LIN {X 0.057,Y -141.322,Z 1092.972,A 0.000,B 0.000,C 90.000,E1 174.894} C_DIS
LIN {X 0.015,Y -142.680,Z 1092.956,A 0.000,B 0.000,C 90.000,E1 172.129} C_DIS
LIN {X -0.005,Y -145.037,Z 1092.931,A 0.000,B 0.000,C 90.000,E1 167.521} C_DIS
LIN {X -0.048,Y -147.662,Z 1092.910,A 0.000,B 0.000,C 90.000,E1 163.866} C_DIS
LIN {X 0.027,Y -150.303,Z 1092.890,A 0.000,B 0.000,C 90.000,E1 160.188} C_DIS
LIN {X 0.039,Y -153.712,Z 1092.870,A 0.000,B 0.000,C 90.000,E1 156.561} C_DIS
LIN {X -0.048,Y -157.126,Z 1092.850,A 0.000,B 0.000,C 90.000,E1 152.999} C_DIS
LIN {X 0.028,Y -161.272,Z 1092.830,A 0.000,B 0.000,C 90.000,E1 149.410} C_DIS
LIN {X 0.046,Y -164.389,Z 1092.815,A 0.000,B 0.000,C 90.000,E1 146.755} C_DIS
LIN {X 0.044,Y -169.066,Z 1092.796,A 0.000,B 0.000,C 90.000,E1 143.256} C_DIS
LIN {X -0.006,Y -171.625,Z 1092.786,A 0.000,B 0.000,C 90.000,E1 141.537} C_DIS
LIN {X 0.042,Y -176.584,Z 1092.767,A 0.000,B 0.000,C 90.000,E1 138.081} C_DIS
LIN {X -0.085,Y -180.882,Z 1092.753,A 0.000,B 0.000,C 90.000,E1 135.567} C_DIS
LIN {X 0.036,Y -186.297,Z 1092.734,A 0.000,B 0.000,C 90.000,E1 132.162} C_DIS
LIN {X 0.103,Y -190.932,Z 1092.720,A 0.000,B 0.000,C 90.000,E1 129.644} C_DIS
LIN {X 0.024,Y -196.700,Z 1092.702,A 0.000,B 0.000,C 90.000,E1 126.377} C_DIS
LIN {X 0.038,Y -199.887,Z 1092.693,A 0.000,B 0.000,C 90.000,E1 124.771} C_DIS
LIN {X 0.020,Y -307.815,Z 1092.693,A 0.000,B 0.000,C 90.000,E1 124.771} C_DIS
LIN {X 0.085,Y -309.073,Z 1092.693,A 0.000,B 0.000,C 90.000,E1 124.739} C_DIS
LIN {X 0.065,Y -312.481,Z 1092.692,A 0.000,B 0.000,C 90.000,E1 124.612} C_DIS
LIN {X -0.118,Y -315.790,Z 1092.691,A 0.000,B 0.000,C 90.000,E1 124.405} C_DIS
LIN {X -0.220,Y -319.464,Z 1092.689,A 0.000,B 0.000,C 90.000,E1 123.992} C_DIS
LIN {X 0.064,Y -321.338,Z 1092.687,A 0.000,B 0.000,C 90.000,E1 123.627} C_DIS
LIN {X 0.172,Y -322.799,Z 1092.685,A 0.000,B 0.000,C 90.000,E1 123.293} C_DIS
LIN {X -0.124,Y -335.754,Z 1092.666,A 0.000,B 0.000,C 90.000,E1 119.873} C_DIS
LIN {X -0.051,Y -347.795,Z 1092.650,A 0.000,B 0.000,C 90.000,E1 117.078} C_DIS
LIN {X 0.064,Y -361.305,Z 1092.635,A 0.000,B 0.000,C 90.000,E1 114.335} C_DIS
LIN {X 0.017,Y -374.646,Z 1092.622,A 0.000,B 0.000,C 90.000,E1 111.972} C_DIS
LIN {X 0.165,Y -389.338,Z 1092.609,A 0.000,B 0.000,C 90.000,E1 109.631} C_DIS
LIN {X -0.088,Y -405.484,Z 1092.597,A 0.000,B 0.000,C 90.000,E1 107.402} C_DIS
LIN {X -0.070,Y -423.198,Z 1092.584,A 0.000,B 0.000,C 90.000,E1 105.190} C_DIS
LIN {X -0.196,Y -442.533,Z 1092.572,A 0.000,B 0.000,C 90.000,E1 103.063} C_DIS
LIN {X -0.226,Y -462.723,Z 1092.561,A 0.000,B 0.000,C 90.000,E1 101.074} C_DIS
LIN {X -0.229,Y -467.843,Z 1092.559,A 0.000,B 0.000,C 90.000,E1 100.602} C_DIS
LIN {X 0.250,Y -469.933,Z 1092.557,A 0.000,B 0.000,C 90.000,E1 100.310} C_DIS
LIN {X 0.102,Y -471.641,Z 1092.556,A 0.000,B 0.000,C 90.000,E1 100.074} C_DIS
LIN {X -0.131,Y -472.922,Z 1092.555,A 0.000,B 0.000,C 90.000,E1 99.849} C_DIS
LIN {X 0.053,Y -474.510,Z 1092.552,A 0.000,B 0.000,C 90.000,E1 99.321} C_DIS
LIN {X 0.169,Y -475.044,Z 1092.549,A 0.000,B 0.000,C 90.000,E1 98.803} C_DIS
LIN {X -0.173,Y -474.615,Z 1092.546,A 0.000,B 0.000,C 90.000,E1 98.341} C_DIS
LIN {X 0.024,Y -473.158,Z 1092.543,A 0.000,B 0.000,C 90.000,E1 97.814} C_DIS
LIN {X -0.177,Y -471.971,Z 1092.542,A 0.000,B 0.000,C 90.000,E1 97.587} C_DIS
LIN {X 0.151,Y -470.390,Z 1092.541,A 0.000,B 0.000,C 90.000,E1 97.296} C_DIS
LIN {X 0.015,Y -455.963,Z 1092.529,A 0.000,B 0.000,C 90.000,E1 95.277} C_DIS
LIN {X 0.138,Y -440.045,Z 1092.516,A 0.000,B 0.000,C 90.000,E1 92.922} C_DIS
LIN {X -0.173,Y -425.406,Z 1092.503,A 0.000,B 0.000,C 90.000,E1 90.573} C_DIS
LIN {X -0.171,Y -407.328,Z 1092.485,A 0.000,B 0.000,C 90.000,E1 87.306} C_DIS
LIN {X -0.175,Y -398.359,Z 1092.476,A 0.000,B 0.000,C 90.000,E1 85.641} C_DIS
LIN {X 0.090,Y -387.622,Z 1092.465,A 0.000,B 0.000,C 90.000,E1 83.628} C_DIS
LIN {X -0.182,Y -378.481,Z 1092.455,A 0.000,B 0.000,C 90.000,E1 81.951} C_DIS
LIN {X 0.185,Y -369.021,Z 1092.445,A 0.000,B 0.000,C 90.000,E1 80.151} C_DIS
LIN {X 0.006,Y -359.223,Z 1092.436,A 0.000,B 0.000,C 90.000,E1 78.409} C_DIS
LIN {X 0.076,Y -347.609,Z 1092.424,A 0.000,B 0.000,C 90.000,E1 76.297} C_DIS
LIN {X -0.043,Y -334.390,Z 1092.410,A 0.000,B 0.000,C 90.000,E1 73.866} C_DIS
LIN {X -0.026,Y -320.149,Z 1092.395,A 0.000,B 0.000,C 90.000,E1 71.040} C_DIS
LIN {X 0.120,Y -305.310,Z 1092.377,A 0.000,B 0.000,C 90.000,E1 67.794} C_DIS
LIN {X -0.115,Y -295.411,Z 1092.364,A 0.000,B 0.000,C 90.000,E1 65.537} C_DIS
LIN {X 0.057,Y -284.299,Z 1092.349,A 0.000,B 0.000,C 90.000,E1 62.820} C_DIS
LIN {X -0.108,Y -274.790,Z 1092.336,A 0.000,B 0.000,C 90.000,E1 60.461} C_DIS
LIN {X -0.125,Y -262.917,Z 1092.318,A 0.000,B 0.000,C 90.000,E1 57.327} C_DIS
LIN {X 0.080,Y -251.527,Z 1092.301,A 0.000,B 0.000,C 90.000,E1 54.069} C_DIS
LIN {X 0.007,Y -240.801,Z 1092.282,A 0.000,B 0.000,C 90.000,E1 50.803} C_DIS
LIN {X -0.042,Y -231.962,Z 1092.266,A 0.000,B 0.000,C 90.000,E1 47.838} C_DIS
LIN {X 0.025,Y -223.685,Z 1092.249,A 0.000,B 0.000,C 90.000,E1 44.798} C_DIS
LIN {X -0.112,Y -215.715,Z 1092.232,A 0.000,B 0.000,C 90.000,E1 41.757} C_DIS
LIN {X 0.040,Y -208.167,Z 1092.214,A 0.000,B 0.000,C 90.000,E1 38.588} C_DIS
LIN {X -0.063,Y -201.049,Z 1092.197,A 0.000,B 0.000,C 90.000,E1 35.438} C_DIS
LIN {X -0.068,Y -194.585,Z 1092.179,A 0.000,B 0.000,C 90.000,E1 32.212} C_DIS
LIN {X -0.104,Y -188.761,Z 1092.161,A 0.000,B 0.000,C 90.000,E1 28.949} C_DIS
LIN {X 0.028,Y -183.659,Z 1092.142,A 0.000,B 0.000,C 90.000,E1 25.591} C_DIS
LIN {X -0.041,Y -179.294,Z 1092.124,A 0.000,B 0.000,C 90.000,E1 22.259} C_DIS
LIN {X 0.017,Y -174.739,Z 1092.100,A 0.000,B 0.000,C 90.000,E1 18.000} C_DIS
LIN {X 0.020,Y -171.298,Z 1092.076,A 0.000,B 0.000,C 90.000,E1 13.716} C_DIS
LIN {X -0.076,Y -168.460,Z 1092.047,A 0.000,B 0.000,C 90.000,E1 8.568} C_DIS
LIN {X -0.045,Y -169.289,Z 1091.949,A 0.000,B 0.000,C 90.000,E1 350.849} C_DIS
LIN {X -0.036,Y -171.949,Z 1091.925,A 0.000,B 0.000,C 90.000,E1 346.520} C_DIS
LIN {X 0.093,Y -175.713,Z 1091.901,A 0.000,B 0.000,C 90.000,E1 342.181} C_DIS
LIN {X 0.092,Y -179.455,Z 1091.882,A 0.000,B 0.000,C 90.000,E1 338.773} C_DIS
LIN {X 0.047,Y -183.849,Z 1091.863,A 0.000,B 0.000,C 90.000,E1 335.409} C_DIS
LIN {X -0.078,Y -188.977,Z 1091.845,A 0.000,B 0.000,C 90.000,E1 332.103} C_DIS
LIN {X -0.056,Y -194.924,Z 1091.827,A 0.000,B 0.000,C 90.000,E1 328.791} C_DIS
LIN {X -0.006,Y -201.529,Z 1091.808,A 0.000,B 0.000,C 90.000,E1 325.515} C_DIS
LIN {X 0.110,Y -208.968,Z 1091.791,A 0.000,B 0.000,C 90.000,E1 322.271} C_DIS
LIN {X -0.059,Y -218.189,Z 1091.771,A 0.000,B 0.000,C 90.000,E1 318.771} C_DIS
LIN {X 0.065,Y -227.268,Z 1091.754,A 0.000,B 0.000,C 90.000,E1 315.648} C_DIS
LIN {X -0.024,Y -236.122,Z 1091.739,A 0.000,B 0.000,C 90.000,E1 313.014} C_DIS
LIN {X 0.104,Y -246.133,Z 1091.724,A 0.000,B 0.000,C 90.000,E1 310.378} C_DIS
LIN {X -0.053,Y -255.734,Z 1091.712,A 0.000,B 0.000,C 90.000,E1 308.222} C_DIS
LIN {X -0.027,Y -269.863,Z 1091.696,A 0.000,B 0.000,C 90.000,E1 305.358} C_DIS
LIN {X 0.093,Y -287.258,Z 1091.679,A 0.000,B 0.000,C 90.000,E1 302.212} C_DIS
LIN {X 0.037,Y -306.101,Z 1091.662,A 0.000,B 0.000,C 90.000,E1 299.205} C_DIS
LIN {X 0.065,Y -326.741,Z 1091.646,A 0.000,B 0.000,C 90.000,E1 296.283} C_DIS
LIN {X 0.009,Y -339.169,Z 1091.637,A 0.000,B 0.000,C 90.000,E1 294.719} C_DIS
LIN {X 0.041,Y -360.003,Z 1091.624,A 0.000,B 0.000,C 90.000,E1 292.386} C_DIS
LIN {X -0.148,Y -373.382,Z 1091.617,A 0.000,B 0.000,C 90.000,E1 291.099} C_DIS
LIN {X 0.075,Y -395.207,Z 1091.606,A 0.000,B 0.000,C 90.000,E1 289.141} C_DIS
LIN {X 0.117,Y -408.891,Z 1091.600,A 0.000,B 0.000,C 90.000,E1 287.946} C_DIS
LIN {X 0.153,Y -419.515,Z 1091.594,A 0.000,B 0.000,C 90.000,E1 286.985} C_DIS
LIN {X -0.054,Y -429.801,Z 1091.589,A 0.000,B 0.000,C 90.000,E1 286.024} C_DIS
LIN {X 0.018,Y -437.221,Z 1091.585,A 0.000,B 0.000,C 90.000,E1 285.245} C_DIS
LIN {X -0.187,Y -444.337,Z 1091.580,A 0.000,B 0.000,C 90.000,E1 284.481} C_DIS
LIN {X 0.162,Y -450.962,Z 1091.576,A 0.000,B 0.000,C 90.000,E1 283.647} C_DIS
LIN {X 0.031,Y -456.996,Z 1091.572,A 0.000,B 0.000,C 90.000,E1 282.883} C_DIS
LIN {X -0.055,Y -462.332,Z 1091.567,A 0.000,B 0.000,C 90.000,E1 282.119} C_DIS
LIN {X -0.183,Y -466.907,Z 1091.563,A 0.000,B 0.000,C 90.000,E1 281.366} C_DIS
LIN {X -0.182,Y -470.757,Z 1091.559,A 0.000,B 0.000,C 90.000,E1 280.602} C_DIS
LIN {X -0.009,Y -472.971,Z 1091.556,A 0.000,B 0.000,C 90.000,E1 280.074} C_DIS
LIN {X 0.097,Y -474.872,Z 1091.553,A 0.000,B 0.000,C 90.000,E1 279.557} C_DIS
LIN {X -0.181,Y -476.497,Z 1091.550,A 0.000,B 0.000,C 90.000,E1 279.086} C_DIS
LIN {X -0.055,Y -477.911,Z 1091.548,A 0.000,B 0.000,C 90.000,E1 278.568} C_DIS
LIN {X 0.084,Y -479.098,Z 1091.545,A 0.000,B 0.000,C 90.000,E1 278.049} C_DIS
LIN {X -0.241,Y -480.072,Z 1091.542,A 0.000,B 0.000,C 90.000,E1 277.587} C_DIS
LIN {X -0.084,Y -480.831,Z 1091.539,A 0.000,B 0.000,C 90.000,E1 277.068} C_DIS
LIN {X 0.082,Y -481.355,Z 1091.536,A 0.000,B 0.000,C 90.000,E1 276.549} C_DIS
LIN {X -0.228,Y -481.615,Z 1091.534,A 0.000,B 0.000,C 90.000,E1 276.087} C_DIS
LIN {X -0.056,Y -481.553,Z 1091.531,A 0.000,B 0.000,C 90.000,E1 275.568} C_DIS
LIN {X 0.117,Y -481.098,Z 1091.528,A 0.000,B 0.000,C 90.000,E1 275.049} C_DIS
LIN {X -0.193,Y -480.276,Z 1091.525,A 0.000,B 0.000,C 90.000,E1 274.588} C_DIS
LIN {X -0.062,Y -478.985,Z 1091.523,A 0.000,B 0.000,C 90.000,E1 274.073} C_DIS
LIN {X 0.098,Y -477.159,Z 1091.520,A 0.000,B 0.000,C 90.000,E1 273.555} C_DIS
LIN {X 0.246,Y -474.669,Z 1091.517,A 0.000,B 0.000,C 90.000,E1 273.037} C_DIS
LIN {X -0.122,Y -471.396,Z 1091.514,A 0.000,B 0.000,C 90.000,E1 272.579} C_DIS
LIN {X -0.030,Y -467.165,Z 1091.511,A 0.000,B 0.000,C 90.000,E1 272.064} C_DIS
LIN {X 0.055,Y -461.872,Z 1091.509,A 0.000,B 0.000,C 90.000,E1 271.547} C_DIS
LIN {X -0.021,Y -455.774,Z 1091.506,A 0.000,B 0.000,C 90.000,E1 271.088} C_DIS
LIN {X -0.052,Y -449.233,Z 1091.504,A 0.000,B 0.000,C 90.000,E1 270.688} C_DIS
LIN {X -0.055,Y -442.292,Z 1091.502,A 0.000,B 0.000,C 90.000,E1 270.344} C_DIS
LIN {X -0.028,Y -434.927,Z 1091.500,A 0.000,B 0.000,C 90.000,E1 270.057} C_DIS
LIN {X 0.026,Y -427.274,Z 1091.499,A 0.000,B 0.000,C 90.000,E1 269.828} C_DIS
LIN {X -0.022,Y -415.947,Z 1091.498,A 0.000,B 0.000,C 90.000,E1 269.599} C_DIS
LIN {X -0.029,Y -407.463,Z 1091.497,A 0.000,B 0.000,C 90.000,E1 269.484} C_DIS
LIN {X 0.170,Y -396.515,Z 1091.497,A 0.000,B 0.000,C 90.000,E1 269.370} C_DIS
LIN {X 0.043,Y -391.580,Z 1091.497,A 0.000,B 0.000,C 90.000,E1 269.370} C_DIS
LIN {X -0.009,Y -181.405,Z 1091.496,A 0.000,B 0.000,C 90.000,E1 269.370} C_DIS
LIN {X -0.068,Y -180.810,Z 1091.471,A 0.000,B 0.000,C 90.000,E1 264.837} C_DIS
LIN {X 0.008,Y -178.912,Z 1091.443,A 0.000,B 0.000,C 90.000,E1 259.746} C_DIS
LIN {X 0.089,Y -175.956,Z 1091.415,A 0.000,B 0.000,C 90.000,E1 254.629} C_DIS
LIN {X 0.035,Y -175.426,Z 1091.410,A 0.000,B 0.000,C 90.000,E1 253.795} C_DIS
LIN {X 0.037,Y -172.186,Z 1091.386,A 0.000,B 0.000,C 90.000,E1 249.518} C_DIS
LIN {X 0.014,Y -171.658,Z 1091.381,A 0.000,B 0.000,C 90.000,E1 248.666} C_DIS
LIN {X -0.003,Y -167.882,Z 1091.358,A 0.000,B 0.000,C 90.000,E1 244.357} C_DIS
LIN {X 0.013,Y -166.619,Z 1091.348,A 0.000,B 0.000,C 90.000,E1 242.615} C_DIS
LIN {X 0.007,Y -162.606,Z 1091.324,A 0.000,B 0.000,C 90.000,E1 238.250} C_DIS
LIN {X -0.019,Y -161.291,Z 1091.314,A 0.000,B 0.000,C 90.000,E1 236.501} C_DIS
LIN {X 0.016,Y -157.290,Z 1091.289,A 0.000,B 0.000,C 90.000,E1 232.065} C_DIS
LIN {X 0.038,Y -156.007,Z 1091.279,A 0.000,B 0.000,C 90.000,E1 230.275} C_DIS
LIN {X -0.002,Y -152.265,Z 1091.255,A 0.000,B 0.000,C 90.000,E1 225.810} C_DIS
LIN {X 0.020,Y -150.503,Z 1091.240,A 0.000,B 0.000,C 90.000,E1 223.095} C_DIS
LIN {X 0.049,Y -147.227,Z 1091.214,A 0.000,B 0.000,C 90.000,E1 218.543} C_DIS
LIN {X 0.019,Y -145.250,Z 1091.194,A 0.000,B 0.000,C 90.000,E1 214.898} C_DIS
LIN {X -0.065,Y -142.366,Z 1091.163,A 0.000,B 0.000,C 90.000,E1 209.411} C_DIS
LIN {X 0.056,Y -141.751,Z 1091.153,A 0.000,B 0.000,C 90.000,E1 207.513} C_DIS
LIN {X -0.019,Y -139.494,Z 1091.117,A 0.000,B 0.000,C 90.000,E1 201.046} C_DIS
LIN {X 0.019,Y -138.999,Z 1091.101,A 0.000,B 0.000,C 90.000,E1 198.236} C_DIS
LIN {X -0.024,Y -138.337,Z 1091.055,A 0.000,B 0.000,C 90.000,E1 189.849} C_DIS
LIN {X -0.003,Y -139.411,Z 1091.008,A 0.000,B 0.000,C 90.000,E1 181.432} C_DIS
LIN {X 0.051,Y -141.323,Z 1090.972,A 0.000,B 0.000,C 90.000,E1 174.894} C_DIS
LIN {X 0.008,Y -142.681,Z 1090.956,A 0.000,B 0.000,C 90.000,E1 172.129} C_DIS
LIN {X -0.012,Y -145.038,Z 1090.931,A 0.000,B 0.000,C 90.000,E1 167.521} C_DIS
LIN {X -0.055,Y -147.664,Z 1090.910,A 0.000,B 0.000,C 90.000,E1 163.866} C_DIS
LIN {X 0.021,Y -150.304,Z 1090.890,A 0.000,B 0.000,C 90.000,E1 160.188} C_DIS
LIN {X 0.032,Y -153.715,Z 1090.870,A 0.000,B 0.000,C 90.000,E1 156.561} C_DIS
LIN {X -0.054,Y -157.129,Z 1090.850,A 0.000,B 0.000,C 90.000,E1 152.999} C_DIS
LIN {X 0.021,Y -161.274,Z 1090.830,A 0.000,B 0.000,C 90.000,E1 149.410} C_DIS
LIN {X 0.039,Y -164.392,Z 1090.815,A 0.000,B 0.000,C 90.000,E1 146.755} C_DIS
LIN {X 0.036,Y -169.069,Z 1090.796,A 0.000,B 0.000,C 90.000,E1 143.256} C_DIS
LIN {X -0.013,Y -171.629,Z 1090.786,A 0.000,B 0.000,C 90.000,E1 141.537} C_DIS
LIN {X 0.035,Y -176.588,Z 1090.767,A 0.000,B 0.000,C 90.000,E1 138.081} C_DIS
LIN {X -0.092,Y -180.886,Z 1090.753,A 0.000,B 0.000,C 90.000,E1 135.567} C_DIS
LIN {X 0.028,Y -186.301,Z 1090.734,A 0.000,B 0.000,C 90.000,E1 132.162} C_DIS
LIN {X 0.095,Y -190.935,Z 1090.720,A 0.000,B 0.000,C 90.000,E1 129.644} C_DIS
LIN {X 0.016,Y -196.704,Z 1090.702,A 0.000,B 0.000,C 90.000,E1 126.377} C_DIS
LIN {X -0.001,Y -199.813,Z 1090.693,A 0.000,B 0.000,C 90.000,E1 124.818} C_DIS
LIN {X -0.037,Y -307.525,Z 1090.693,A 0.000,B 0.000,C 90.000,E1 124.818} C_DIS
LIN {X 0.073,Y -310.213,Z 1090.693,A 0.000,B 0.000,C 90.000,E1 124.739} C_DIS
LIN {X -0.034,Y -313.199,Z 1090.692,A 0.000,B 0.000,C 90.000,E1 124.612} C_DIS
LIN {X -0.131,Y -316.798,Z 1090.691,A 0.000,B 0.000,C 90.000,E1 124.326} C_DIS
LIN {X 0.153,Y -320.409,Z 1090.688,A 0.000,B 0.000,C 90.000,E1 123.785} C_DIS
LIN {X -0.044,Y -322.074,Z 1090.686,A 0.000,B 0.000,C 90.000,E1 123.499} C_DIS
LIN {X 0.117,Y -324.479,Z 1090.682,A 0.000,B 0.000,C 90.000,E1 122.832} C_DIS
LIN {X 0.079,Y -335.078,Z 1090.667,A 0.000,B 0.000,C 90.000,E1 120.001} C_DIS
LIN {X -0.167,Y -347.036,Z 1090.651,A 0.000,B 0.000,C 90.000,E1 117.257} C_DIS
LIN {X -0.091,Y -360.460,Z 1090.636,A 0.000,B 0.000,C 90.000,E1 114.515} C_DIS
LIN {X -0.170,Y -373.717,Z 1090.623,A 0.000,B 0.000,C 90.000,E1 112.153} C_DIS
LIN {X -0.055,Y -388.317,Z 1090.610,A 0.000,B 0.000,C 90.000,E1 109.812} C_DIS
LIN {X 0.164,Y -404.365,Z 1090.597,A 0.000,B 0.000,C 90.000,E1 107.511} C_DIS
LIN {X 0.045,Y -421.975,Z 1090.585,A 0.000,B 0.000,C 90.000,E1 105.315} C_DIS
LIN {X -0.023,Y -441.228,Z 1090.573,A 0.000,B 0.000,C 90.000,E1 103.175} C_DIS
LIN {X -0.142,Y -461.382,Z 1090.562,A 0.000,B 0.000,C 90.000,E1 101.186} C_DIS
LIN {X -0.225,Y -468.893,Z 1090.558,A 0.000,B 0.000,C 90.000,E1 100.489} C_DIS
LIN {X -0.197,Y -470.709,Z 1090.557,A 0.000,B 0.000,C 90.000,E1 100.254} C_DIS
LIN {X 0.120,Y -472.215,Z 1090.555,A 0.000,B 0.000,C 90.000,E1 99.962} C_DIS
LIN {X -0.029,Y -473.339,Z 1090.554,A 0.000,B 0.000,C 90.000,E1 99.726} C_DIS
LIN {X 0.080,Y -474.681,Z 1090.551,A 0.000,B 0.000,C 90.000,E1 99.208} C_DIS
LIN {X 0.200,Y -475.003,Z 1090.548,A 0.000,B 0.000,C 90.000,E1 98.690} C_DIS
LIN {X -0.072,Y -474.361,Z 1090.546,A 0.000,B 0.000,C 90.000,E1 98.219} C_DIS
LIN {X 0.058,Y -472.655,Z 1090.543,A 0.000,B 0.000,C 90.000,E1 97.701} C_DIS
LIN {X -0.082,Y -471.308,Z 1090.541,A 0.000,B 0.000,C 90.000,E1 97.466} C_DIS
LIN {X -0.013,Y -458.786,Z 1090.532,A 0.000,B 0.000,C 90.000,E1 95.682} C_DIS
LIN {X -0.038,Y -440.979,Z 1090.517,A 0.000,B 0.000,C 90.000,E1 93.094} C_DIS
LIN {X 0.100,Y -426.312,Z 1090.504,A 0.000,B 0.000,C 90.000,E1 90.688} C_DIS
LIN {X 0.046,Y -409.623,Z 1090.487,A 0.000,B 0.000,C 90.000,E1 87.707} C_DIS
LIN {X 0.053,Y -400.706,Z 1090.478,A 0.000,B 0.000,C 90.000,E1 86.045} C_DIS
LIN {X -0.042,Y -391.577,Z 1090.469,A 0.000,B 0.000,C 90.000,E1 84.375} C_DIS
LIN {X 0.146,Y -379.320,Z 1090.456,A 0.000,B 0.000,C 90.000,E1 82.064} C_DIS
LIN {X 0.097,Y -369.888,Z 1090.446,A 0.000,B 0.000,C 90.000,E1 80.330} C_DIS
LIN {X 0.003,Y -360.110,Z 1090.437,A 0.000,B 0.000,C 90.000,E1 78.578} C_DIS
LIN {X 0.096,Y -348.480,Z 1090.425,A 0.000,B 0.000,C 90.000,E1 76.464} C_DIS
LIN {X 0.022,Y -336.882,Z 1090.413,A 0.000,B 0.000,C 90.000,E1 74.338} C_DIS
LIN {X -0.039,Y -320.985,Z 1090.396,A 0.000,B 0.000,C 90.000,E1 71.221} C_DIS
LIN {X 0.038,Y -304.647,Z 1090.376,A 0.000,B 0.000,C 90.000,E1 67.667} C_DIS
LIN {X 0.060,Y -294.737,Z 1090.363,A 0.000,B 0.000,C 90.000,E1 65.357} C_DIS
LIN {X 0.082,Y -283.638,Z 1090.348,A 0.000,B 0.000,C 90.000,E1 62.666} C_DIS
LIN {X 0.014,Y -274.117,Z 1090.335,A 0.000,B 0.000,C 90.000,E1 60.284} C_DIS
LIN {X -0.031,Y -263.551,Z 1090.319,A 0.000,B 0.000,C 90.000,E1 57.502} C_DIS
LIN {X 0.027,Y -253.366,Z 1090.304,A 0.000,B 0.000,C 90.000,E1 54.642} C_DIS
LIN {X 0.005,Y -242.470,Z 1090.285,A 0.000,B 0.000,C 90.000,E1 51.376} C_DIS
LIN {X 0.023,Y -233.477,Z 1090.269,A 0.000,B 0.000,C 90.000,E1 48.405} C_DIS
LIN {X -0.046,Y -225.100,Z 1090.252,A 0.000,B 0.000,C 90.000,E1 45.405} C_DIS
LIN {X 0.009,Y -217.053,Z 1090.235,A 0.000,B 0.000,C 90.000,E1 42.324} C_DIS
LIN {X 0.037,Y -209.373,Z 1090.218,A 0.000,B 0.000,C 90.000,E1 39.197} C_DIS
LIN {X 0.089,Y -202.130,Z 1090.200,A 0.000,B 0.000,C 90.000,E1 36.011} C_DIS
LIN {X -0.057,Y -195.547,Z 1090.182,A 0.000,B 0.000,C 90.000,E1 32.832} C_DIS
LIN {X 0.028,Y -189.582,Z 1090.164,A 0.000,B 0.000,C 90.000,E1 29.539} C_DIS
LIN {X 0.015,Y -184.339,Z 1090.146,A 0.000,B 0.000,C 90.000,E1 26.232} C_DIS
LIN {X -0.035,Y -179.835,Z 1090.127,A 0.000,B 0.000,C 90.000,E1 22.898} C_DIS
LIN {X -0.057,Y -175.133,Z 1090.104,A 0.000,B 0.000,C 90.000,E1 18.671} C_DIS
LIN {X 0.051,Y -171.523,Z 1090.080,A 0.000,B 0.000,C 90.000,E1 14.356} C_DIS
LIN {X -0.042,Y -168.521,Z 1090.051,A 0.000,B 0.000,C 90.000,E1 9.208} C_DIS
LIN {X -0.052,Y -166.625,Z 1090.003,A 0.000,B 0.000,C 90.000,E1 0.516} C_DIS
LIN {X -0.075,Y -168.283,Z 1089.959,A 0.000,B 0.000,C 90.000,E1 352.591} C_DIS
LIN {X 0.032,Y -171.107,Z 1089.930,A 0.000,B 0.000,C 90.000,E1 347.353} C_DIS
LIN {X -0.086,Y -174.643,Z 1089.906,A 0.000,B 0.000,C 90.000,E1 343.087} C_DIS
LIN {X -0.012,Y -178.234,Z 1089.887,A 0.000,B 0.000,C 90.000,E1 339.645} C_DIS
LIN {X 0.073,Y -182.483,Z 1089.868,A 0.000,B 0.000,C 90.000,E1 336.230} C_DIS
LIN {X 0.086,Y -187.395,Z 1089.849,A 0.000,B 0.000,C 90.000,E1 332.871} C_DIS
LIN {X -0.020,Y -193.155,Z 1089.831,A 0.000,B 0.000,C 90.000,E1 329.587} C_DIS
LIN {X 0.046,Y -199.661,Z 1089.813,A 0.000,B 0.000,C 90.000,E1 326.294} C_DIS
LIN {X 0.112,Y -206.915,Z 1089.795,A 0.000,B 0.000,C 90.000,E1 323.050} C_DIS
LIN {X -0.096,Y -215.914,Z 1089.775,A 0.000,B 0.000,C 90.000,E1 319.542} C_DIS
LIN {X -0.035,Y -224.765,Z 1089.758,A 0.000,B 0.000,C 90.000,E1 316.419} C_DIS
LIN {X -0.071,Y -234.681,Z 1089.741,A 0.000,B 0.000,C 90.000,E1 313.380} C_DIS
LIN {X 0.013,Y -244.501,Z 1089.726,A 0.000,B 0.000,C 90.000,E1 310.744} C_DIS
LIN {X 0.018,Y -253.949,Z 1089.714,A 0.000,B 0.000,C 90.000,E1 308.543} C_DIS
LIN {X 0.011,Y -267.943,Z 1089.698,A 0.000,B 0.000,C 90.000,E1 305.678} C_DIS
LIN {X 0.010,Y -285.219,Z 1089.681,A 0.000,B 0.000,C 90.000,E1 302.546} C_DIS
LIN {X -0.119,Y -303.961,Z 1089.664,A 0.000,B 0.000,C 90.000,E1 299.539} C_DIS
LIN {X -0.154,Y -324.398,Z 1089.648,A 0.000,B 0.000,C 90.000,E1 296.616} C_DIS
LIN {X -0.086,Y -336.625,Z 1089.639,A 0.000,B 0.000,C 90.000,E1 295.027} C_DIS
LIN {X 0.158,Y -354.884,Z 1089.627,A 0.000,B 0.000,C 90.000,E1 292.898} C_DIS
LIN {X 0.031,Y -370.301,Z 1089.619,A 0.000,B 0.000,C 90.000,E1 291.354} C_DIS
LIN {X -0.209,Y -394.793,Z 1089.607,A 0.000,B 0.000,C 90.000,E1 289.214} C_DIS
LIN {X 0.004,Y -408.437,Z 1089.600,A 0.000,B 0.000,C 90.000,E1 288.000} C_DIS
LIN {X 0.063,Y -419.061,Z 1089.595,A 0.000,B 0.000,C 90.000,E1 287.040} C_DIS
LIN {X -0.119,Y -429.322,Z 1089.589,A 0.000,B 0.000,C 90.000,E1 286.079} C_DIS
LIN {X -0.026,Y -436.754,Z 1089.585,A 0.000,B 0.000,C 90.000,E1 285.300} C_DIS
LIN {X -0.156,Y -443.847,Z 1089.581,A 0.000,B 0.000,C 90.000,E1 284.537} C_DIS
LIN {X 0.080,Y -450.518,Z 1089.576,A 0.000,B 0.000,C 90.000,E1 283.716} C_DIS
LIN {X 0.050,Y -456.624,Z 1089.572,A 0.000,B 0.000,C 90.000,E1 282.939} C_DIS
LIN {X -0.039,Y -462.039,Z 1089.568,A 0.000,B 0.000,C 90.000,E1 282.175} C_DIS
LIN {X -0.171,Y -466.664,Z 1089.563,A 0.000,B 0.000,C 90.000,E1 281.422} C_DIS
LIN {X -0.174,Y -470.586,Z 1089.559,A 0.000,B 0.000,C 90.000,E1 280.658} C_DIS
LIN {X -0.085,Y -472.840,Z 1089.556,A 0.000,B 0.000,C 90.000,E1 280.141} C_DIS
LIN {X 0.102,Y -474.769,Z 1089.553,A 0.000,B 0.000,C 90.000,E1 279.613} C_DIS
LIN {X -0.253,Y -476.432,Z 1089.551,A 0.000,B 0.000,C 90.000,E1 279.151} C_DIS
LIN {X -0.053,Y -477.877,Z 1089.548,A 0.000,B 0.000,C 90.000,E1 278.624} C_DIS
LIN {X 0.086,Y -479.117,Z 1089.545,A 0.000,B 0.000,C 90.000,E1 278.106} C_DIS
LIN {X -0.241,Y -480.117,Z 1089.542,A 0.000,B 0.000,C 90.000,E1 277.644} C_DIS
LIN {X 0.081,Y -481.521,Z 1089.537,A 0.000,B 0.000,C 90.000,E1 276.606} C_DIS
LIN {X -0.228,Y -481.827,Z 1089.534,A 0.000,B 0.000,C 90.000,E1 276.144} C_DIS
LIN {X -0.055,Y -481.861,Z 1089.531,A 0.000,B 0.000,C 90.000,E1 275.625} C_DIS
LIN {X 0.117,Y -481.490,Z 1089.528,A 0.000,B 0.000,C 90.000,E1 275.106} C_DIS
LIN {X -0.190,Y -480.746,Z 1089.526,A 0.000,B 0.000,C 90.000,E1 274.645} C_DIS
LIN {X -0.058,Y -479.531,Z 1089.523,A 0.000,B 0.000,C 90.000,E1 274.131} C_DIS
LIN {X 0.105,Y -477.763,Z 1089.520,A 0.000,B 0.000,C 90.000,E1 273.612} C_DIS
LIN {X -0.218,Y -475.356,Z 1089.517,A 0.000,B 0.000,C 90.000,E1 273.151} C_DIS
LIN {X -0.109,Y -472.228,Z 1089.515,A 0.000,B 0.000,C 90.000,E1 272.636} C_DIS
LIN {X -0.013,Y -468.146,Z 1089.512,A 0.000,B 0.000,C 90.000,E1 272.121} C_DIS
LIN {X 0.077,Y -462.994,Z 1089.509,A 0.000,B 0.000,C 90.000,E1 271.604} C_DIS
LIN {X -0.002,Y -460.159,Z 1089.508,A 0.000,B 0.000,C 90.000,E1 271.375} C_DIS
LIN {X 0.124,Y -453.930,Z 1089.505,A 0.000,B 0.000,C 90.000,E1 270.917} C_DIS
LIN {X -0.175,Y -447.393,Z 1089.503,A 0.000,B 0.000,C 90.000,E1 270.573} C_DIS
LIN {X -0.024,Y -440.345,Z 1089.501,A 0.000,B 0.000,C 90.000,E1 270.229} C_DIS
LIN {X 0.151,Y -432.932,Z 1089.500,A 0.000,B 0.000,C 90.000,E1 269.943} C_DIS
LIN {X -0.102,Y -425.067,Z 1089.499,A 0.000,B 0.000,C 90.000,E1 269.771} C_DIS
LIN {X 0.011,Y -417.263,Z 1089.498,A 0.000,B 0.000,C 90.000,E1 269.599} C_DIS
LIN {X -0.034,Y -408.836,Z 1089.497,A 0.000,B 0.000,C 90.000,E1 269.484} C_DIS
LIN {X 0.128,Y -398.132,Z 1089.497,A 0.000,B 0.000,C 90.000,E1 269.370} C_DIS
LIN {X -0.009,Y -393.878,Z 1089.496,A 0.000,B 0.000,C 90.000,E1 269.370} C_DIS
LIN {X -0.035,Y -181.403,Z 1089.496,A 0.000,B 0.000,C 90.000,E1 269.370} C_DIS
LIN {X 0.083,Y -180.807,Z 1089.471,A 0.000,B 0.000,C 90.000,E1 264.780} C_DIS
LIN {X -0.020,Y -178.908,Z 1089.443,A 0.000,B 0.000,C 90.000,E1 259.746} C_DIS
LIN {X 0.061,Y -175.953,Z 1089.415,A 0.000,B 0.000,C 90.000,E1 254.629} C_DIS
LIN {X 0.008,Y -175.418,Z 1089.410,A 0.000,B 0.000,C 90.000,E1 253.795} C_DIS
LIN {X 0.011,Y -172.180,Z 1089.386,A 0.000,B 0.000,C 90.000,E1 249.518} C_DIS
LIN {X 0.049,Y -171.652,Z 1089.381,A 0.000,B 0.000,C 90.000,E1 248.646} C_DIS
LIN {X 0.043,Y -167.876,Z 1089.358,A 0.000,B 0.000,C 90.000,E1 244.332} C_DIS
LIN {X -0.013,Y -166.611,Z 1089.348,A 0.000,B 0.000,C 90.000,E1 242.615} C_DIS
LIN {X -0.020,Y -162.599,Z 1089.324,A 0.000,B 0.000,C 90.000,E1 238.250} C_DIS
LIN {X -0.046,Y -161.284,Z 1089.314,A 0.000,B 0.000,C 90.000,E1 236.501} C_DIS
LIN {X -0.011,Y -157.282,Z 1089.289,A 0.000,B 0.000,C 90.000,E1 232.065} C_DIS
LIN {X 0.013,Y -156.001,Z 1089.279,A 0.000,B 0.000,C 90.000,E1 230.275} C_DIS
LIN {X -0.027,Y -152.258,Z 1089.254,A 0.000,B 0.000,C 90.000,E1 225.810} C_DIS
LIN {X -0.005,Y -150.497,Z 1089.239,A 0.000,B 0.000,C 90.000,E1 223.095} C_DIS
LIN {X 0.025,Y -147.221,Z 1089.214,A 0.000,B 0.000,C 90.000,E1 218.543} C_DIS
LIN {X -0.005,Y -145.243,Z 1089.194,A 0.000,B 0.000,C 90.000,E1 214.898} C_DIS
LIN {X -0.089,Y -142.362,Z 1089.163,A 0.000,B 0.000,C 90.000,E1 209.411} C_DIS
LIN {X 0.032,Y -141.748,Z 1089.153,A 0.000,B 0.000,C 90.000,E1 207.513} C_DIS
LIN {X -0.041,Y -139.492,Z 1089.117,A 0.000,B 0.000,C 90.000,E1 201.046} C_DIS
LIN {X -0.005,Y -138.996,Z 1089.101,A 0.000,B 0.000,C 90.000,E1 198.236} C_DIS
LIN {X -0.049,Y -138.336,Z 1089.055,A 0.000,B 0.000,C 90.000,E1 189.849} C_DIS
LIN {X -0.026,Y -139.414,Z 1089.008,A 0.000,B 0.000,C 90.000,E1 181.432} C_DIS
LIN {X 0.028,Y -141.327,Z 1088.972,A 0.000,B 0.000,C 90.000,E1 174.894} C_DIS
LIN {X -0.016,Y -142.685,Z 1088.956,A 0.000,B 0.000,C 90.000,E1 172.129} C_DIS
LIN {X -0.036,Y -145.044,Z 1088.931,A 0.000,B 0.000,C 90.000,E1 167.521} C_DIS
LIN {X -0.038,Y -147.670,Z 1088.910,A 0.000,B 0.000,C 90.000,E1 163.850} C_DIS
LIN {X -0.005,Y -150.312,Z 1088.890,A 0.000,B 0.000,C 90.000,E1 160.188} C_DIS
LIN {X 0.007,Y -153.725,Z 1088.870,A 0.000,B 0.000,C 90.000,E1 156.561} C_DIS
LIN {X -0.080,Y -157.138,Z 1088.850,A 0.000,B 0.000,C 90.000,E1 152.999} C_DIS
LIN {X -0.005,Y -161.286,Z 1088.830,A 0.000,B 0.000,C 90.000,E1 149.410} C_DIS
LIN {X 0.012,Y -164.403,Z 1088.815,A 0.000,B 0.000,C 90.000,E1 146.755} C_DIS
LIN {X 0.009,Y -169.083,Z 1088.796,A 0.000,B 0.000,C 90.000,E1 143.256} C_DIS
LIN {X -0.040,Y -171.640,Z 1088.786,A 0.000,B 0.000,C 90.000,E1 141.537} C_DIS
LIN {X 0.007,Y -176.602,Z 1088.767,A 0.000,B 0.000,C 90.000,E1 138.081} C_DIS
LIN {X 0.008,Y -180.900,Z 1088.753,A 0.000,B 0.000,C 90.000,E1 135.526} C_DIS
LIN {X 0.000,Y -186.316,Z 1088.734,A 0.000,B 0.000,C 90.000,E1 132.162} C_DIS
LIN {X 0.067,Y -190.950,Z 1088.720,A 0.000,B 0.000,C 90.000,E1 129.644} C_DIS
LIN {X -0.014,Y -196.720,Z 1088.702,A 0.000,B 0.000,C 90.000,E1 126.377} C_DIS
LIN {X -0.023,Y -199.729,Z 1088.694,A 0.000,B 0.000,C 90.000,E1 124.865} C_DIS
LIN {X 0.181,Y -306.878,Z 1088.694,A 0.000,B 0.000,C 90.000,E1 124.818} C_DIS
LIN {X 0.077,Y -308.475,Z 1088.693,A 0.000,B 0.000,C 90.000,E1 124.818} C_DIS
LIN {X 0.026,Y -311.216,Z 1088.693,A 0.000,B 0.000,C 90.000,E1 124.739} C_DIS
LIN {X 0.037,Y -314.513,Z 1088.692,A 0.000,B 0.000,C 90.000,E1 124.532} C_DIS
LIN {X -0.199,Y -318.162,Z 1088.690,A 0.000,B 0.000,C 90.000,E1 124.199} C_DIS
LIN {X 0.060,Y -321.640,Z 1088.687,A 0.000,B 0.000,C 90.000,E1 123.579} C_DIS
LIN {X -0.133,Y -323.003,Z 1088.685,A 0.000,B 0.000,C 90.000,E1 123.293} C_DIS
LIN {X -0.111,Y -334.676,Z 1088.667,A 0.000,B 0.000,C 90.000,E1 120.129} C_DIS
LIN {X -0.072,Y -346.587,Z 1088.652,A 0.000,B 0.000,C 90.000,E1 117.334} C_DIS
LIN {X 0.007,Y -359.956,Z 1088.637,A 0.000,B 0.000,C 90.000,E1 114.591} C_DIS
LIN {X 0.069,Y -373.163,Z 1088.623,A 0.000,B 0.000,C 90.000,E1 112.206} C_DIS
LIN {X 0.041,Y -387.711,Z 1088.610,A 0.000,B 0.000,C 90.000,E1 109.885} C_DIS
LIN {X -0.126,Y -403.701,Z 1088.598,A 0.000,B 0.000,C 90.000,E1 107.638} C_DIS
LIN {X -0.157,Y -421.249,Z 1088.586,A 0.000,B 0.000,C 90.000,E1 105.426} C_DIS
LIN {X 0.060,Y -440.444,Z 1088.574,A 0.000,B 0.000,C 90.000,E1 103.244} C_DIS
LIN {X -0.005,Y -460.575,Z 1088.563,A 0.000,B 0.000,C 90.000,E1 101.243} C_DIS
LIN {X -0.127,Y -468.224,Z 1088.558,A 0.000,B 0.000,C 90.000,E1 100.546} C_DIS
LIN {X -0.140,Y -470.231,Z 1088.557,A 0.000,B 0.000,C 90.000,E1 100.310} C_DIS
LIN {X -0.155,Y -471.756,Z 1088.556,A 0.000,B 0.000,C 90.000,E1 100.074} C_DIS
LIN {X 0.085,Y -472.988,Z 1088.554,A 0.000,B 0.000,C 90.000,E1 99.792} C_DIS
LIN {X -0.059,Y -473.891,Z 1088.553,A 0.000,B 0.000,C 90.000,E1 99.557} C_DIS
LIN {X 0.132,Y -474.866,Z 1088.550,A 0.000,B 0.000,C 90.000,E1 99.029} C_DIS
LIN {X -0.216,Y -474.859,Z 1088.547,A 0.000,B 0.000,C 90.000,E1 98.568} C_DIS
LIN {X -0.087,Y -473.873,Z 1088.545,A 0.000,B 0.000,C 90.000,E1 98.049} C_DIS
LIN {X 0.044,Y -471.741,Z 1088.542,A 0.000,B 0.000,C 90.000,E1 97.530} C_DIS
LIN {X 0.016,Y -466.489,Z 1088.538,A 0.000,B 0.000,C 90.000,E1 96.777} C_DIS
LIN {X -0.005,Y -453.948,Z 1088.528,A 0.000,B 0.000,C 90.000,E1 94.992} C_DIS
LIN {X -0.099,Y -439.819,Z 1088.516,A 0.000,B 0.000,C 90.000,E1 92.922} C_DIS
LIN {X 0.013,Y -425.222,Z 1088.503,A 0.000,B 0.000,C 90.000,E1 90.516} C_DIS
LIN {X 0.001,Y -407.144,Z 1088.485,A 0.000,B 0.000,C 90.000,E1 87.249} C_DIS
LIN {X -0.011,Y -398.179,Z 1088.475,A 0.000,B 0.000,C 90.000,E1 85.584} C_DIS
LIN {X -0.137,Y -387.422,Z 1088.464,A 0.000,B 0.000,C 90.000,E1 83.628} C_DIS
LIN {X -0.032,Y -378.244,Z 1088.455,A 0.000,B 0.000,C 90.000,E1 81.894} C_DIS
LIN {X -0.038,Y -368.739,Z 1088.445,A 0.000,B 0.000,C 90.000,E1 80.151} C_DIS
LIN {X 0.207,Y -358.932,Z 1088.435,A 0.000,B 0.000,C 90.000,E1 78.342} C_DIS
LIN {X -0.067,Y -347.290,Z 1088.424,A 0.000,B 0.000,C 90.000,E1 76.284} C_DIS
LIN {X 0.147,Y -334.074,Z 1088.410,A 0.000,B 0.000,C 90.000,E1 73.795} C_DIS
LIN {X -0.093,Y -321.429,Z 1088.396,A 0.000,B 0.000,C 90.000,E1 71.329} C_DIS
LIN {X -0.096,Y -305.054,Z 1088.377,A 0.000,B 0.000,C 90.000,E1 67.794} C_DIS
LIN {X -0.067,Y -295.119,Z 1088.364,A 0.000,B 0.000,C 90.000,E1 65.485} C_DIS
LIN {X -0.031,Y -283.999,Z 1088.349,A 0.000,B 0.000,C 90.000,E1 62.794} C_DIS
LIN {X -0.004,Y -273.109,Z 1088.334,A 0.000,B 0.000,C 90.000,E1 60.049} C_DIS
LIN {X 0.020,Y -262.568,Z 1088.318,A 0.000,B 0.000,C 90.000,E1 57.248} C_DIS
LIN {X 0.014,Y -251.174,Z 1088.300,A 0.000,B 0.000,C 90.000,E1 54.036} C_DIS
LIN {X 0.127,Y -240.418,Z 1088.282,A 0.000,B 0.000,C 90.000,E1 50.723} C_DIS
LIN {X 0.033,Y -230.456,Z 1088.263,A 0.000,B 0.000,C 90.000,E1 47.391} C_DIS
LIN {X 0.055,Y -222.182,Z 1088.246,A 0.000,B 0.000,C 90.000,E1 44.352} C_DIS
LIN {X -0.113,Y -214.201,Z 1088.229,A 0.000,B 0.000,C 90.000,E1 41.310} C_DIS
LIN {X -0.127,Y -206.622,Z 1088.212,A 0.000,B 0.000,C 90.000,E1 38.177} C_DIS
LIN {X 0.022,Y -199.619,Z 1088.194,A 0.000,B 0.000,C 90.000,E1 34.945} C_DIS
LIN {X -0.024,Y -193.184,Z 1088.176,A 0.000,B 0.000,C 90.000,E1 31.720} C_DIS
LIN {X -0.026,Y -187.473,Z 1088.158,A 0.000,B 0.000,C 90.000,E1 28.437} C_DIS
LIN {X 0.073,Y -182.507,Z 1088.139,A 0.000,B 0.000,C 90.000,E1 25.079} C_DIS
LIN {X 0.069,Y -178.242,Z 1088.121,A 0.000,B 0.000,C 90.000,E1 21.716} C_DIS
LIN {X -0.062,Y -174.598,Z 1088.102,A 0.000,B 0.000,C 90.000,E1 18.362} C_DIS
LIN {X -0.019,Y -171.070,Z 1088.078,A 0.000,B 0.000,C 90.000,E1 14.064} C_DIS
LIN {X 0.041,Y -168.167,Z 1088.049,A 0.000,B 0.000,C 90.000,E1 8.859} C_DIS
LIN {X -0.031,Y -166.424,Z 1087.997,A 0.000,B 0.000,C 90.000,E1 359.542} C_DIS
LIN {X -0.093,Y -168.408,Z 1087.954,A 0.000,B 0.000,C 90.000,E1 351.724} C_DIS
LIN {X 0.088,Y -171.501,Z 1087.925,A 0.000,B 0.000,C 90.000,E1 346.464} C_DIS
LIN {X 0.035,Y -175.262,Z 1087.901,A 0.000,B 0.000,C 90.000,E1 342.181} C_DIS
LIN {X 0.022,Y -179.041,Z 1087.882,A 0.000,B 0.000,C 90.000,E1 338.773} C_DIS
LIN {X -0.035,Y -183.442,Z 1087.863,A 0.000,B 0.000,C 90.000,E1 335.409} C_DIS
LIN {X 0.084,Y -188.560,Z 1087.845,A 0.000,B 0.000,C 90.000,E1 332.025} C_DIS
LIN {X 0.004,Y -194.541,Z 1087.826,A 0.000,B 0.000,C 90.000,E1 328.742} C_DIS
LIN {X 0.040,Y -201.253,Z 1087.808,A 0.000,B 0.000,C 90.000,E1 325.468} C_DIS
LIN {X -0.023,Y -208.711,Z 1087.790,A 0.000,B 0.000,C 90.000,E1 322.271} C_DIS
LIN {X 0.097,Y -217.877,Z 1087.771,A 0.000,B 0.000,C 90.000,E1 318.690} C_DIS
LIN {X -0.102,Y -227.017,Z 1087.753,A 0.000,B 0.000,C 90.000,E1 315.648} C_DIS
LIN {X -0.041,Y -235.904,Z 1087.739,A 0.000,B 0.000,C 90.000,E1 312.975} C_DIS
LIN {X -0.088,Y -245.865,Z 1087.724,A 0.000,B 0.000,C 90.000,E1 310.378} C_DIS
LIN {X -0.057,Y -255.515,Z 1087.712,A 0.000,B 0.000,C 90.000,E1 308.177} C_DIS
LIN {X 0.063,Y -267.845,Z 1087.698,A 0.000,B 0.000,C 90.000,E1 305.644} C_DIS
LIN {X -0.103,Y -285.173,Z 1087.681,A 0.000,B 0.000,C 90.000,E1 302.546} C_DIS
LIN {X 0.024,Y -303.957,Z 1087.664,A 0.000,B 0.000,C 90.000,E1 299.489} C_DIS
LIN {X 0.075,Y -322.069,Z 1087.649,A 0.000,B 0.000,C 90.000,E1 296.873} C_DIS
LIN {X 0.103,Y -334.139,Z 1087.641,A 0.000,B 0.000,C 90.000,E1 295.283} C_DIS
LIN {X 0.090,Y -349.711,Z 1087.630,A 0.000,B 0.000,C 90.000,E1 293.462} C_DIS
LIN {X 0.061,Y -365.161,Z 1087.621,A 0.000,B 0.000,C 90.000,E1 291.844} C_DIS
LIN {X -0.065,Y -384.605,Z 1087.611,A 0.000,B 0.000,C 90.000,E1 290.066} C_DIS
LIN {X -0.075,Y -401.072,Z 1087.604,A 0.000,B 0.000,C 90.000,E1 288.652} C_DIS
LIN {X -0.018,Y -414.623,Z 1087.597,A 0.000,B 0.000,C 90.000,E1 287.457} C_DIS
LIN {X 0.013,Y -422.423,Z 1087.593,A 0.000,B 0.000,C 90.000,E1 286.732} C_DIS
LIN {X 0.092,Y -432.635,Z 1087.587,A 0.000,B 0.000,C 90.000,E1 285.717} C_DIS
LIN {X 0.151,Y -439.769,Z 1087.583,A 0.000,B 0.000,C 90.000,E1 284.954} C_DIS
LIN {X -0.124,Y -446.387,Z 1087.579,A 0.000,B 0.000,C 90.000,E1 284.245} C_DIS
LIN {X 0.056,Y -454.896,Z 1087.573,A 0.000,B 0.000,C 90.000,E1 283.175} C_DIS
LIN {X -0.042,Y -460.545,Z 1087.569,A 0.000,B 0.000,C 90.000,E1 282.411} C_DIS
LIN {X -0.193,Y -465.444,Z 1087.565,A 0.000,B 0.000,C 90.000,E1 281.658} C_DIS
LIN {X -0.201,Y -469.550,Z 1087.560,A 0.000,B 0.000,C 90.000,E1 280.894} C_DIS
LIN {X -0.264,Y -473.002,Z 1087.556,A 0.000,B 0.000,C 90.000,E1 280.141} C_DIS
LIN {X -0.077,Y -474.940,Z 1087.553,A 0.000,B 0.000,C 90.000,E1 279.613} C_DIS
LIN {X 0.039,Y -476.611,Z 1087.551,A 0.000,B 0.000,C 90.000,E1 279.095} C_DIS
LIN {X 0.242,Y -478.053,Z 1087.548,A 0.000,B 0.000,C 90.000,E1 278.568} C_DIS
LIN {X -0.092,Y -479.290,Z 1087.545,A 0.000,B 0.000,C 90.000,E1 278.106} C_DIS
LIN {X 0.218,Y -481.145,Z 1087.539,A 0.000,B 0.000,C 90.000,E1 277.068} C_DIS
LIN {X -0.094,Y -481.762,Z 1087.537,A 0.000,B 0.000,C 90.000,E1 276.606} C_DIS
LIN {X 0.077,Y -482.110,Z 1087.534,A 0.000,B 0.000,C 90.000,E1 276.087} C_DIS
LIN {X -0.228,Y -482.115,Z 1087.531,A 0.000,B 0.000,C 90.000,E1 275.625} C_DIS
LIN {X -0.053,Y -481.785,Z 1087.528,A 0.000,B 0.000,C 90.000,E1 275.106} C_DIS
LIN {X 0.120,Y -481.050,Z 1087.526,A 0.000,B 0.000,C 90.000,E1 274.588} C_DIS
LIN {X -0.225,Y -479.812,Z 1087.523,A 0.000,B 0.000,C 90.000,E1 274.131} C_DIS
LIN {X -0.059,Y -478.040,Z 1087.520,A 0.000,B 0.000,C 90.000,E1 273.612} C_DIS
LIN {X 0.094,Y -475.592,Z 1087.517,A 0.000,B 0.000,C 90.000,E1 273.094} C_DIS
LIN {X 0.204,Y -472.444,Z 1087.515,A 0.000,B 0.000,C 90.000,E1 272.579} C_DIS
LIN {X -0.170,Y -468.333,Z 1087.512,A 0.000,B 0.000,C 90.000,E1 272.121} C_DIS
LIN {X -0.077,Y -463.172,Z 1087.509,A 0.000,B 0.000,C 90.000,E1 271.604} C_DIS
LIN {X -0.155,Y -460.354,Z 1087.508,A 0.000,B 0.000,C 90.000,E1 271.375} C_DIS
LIN {X -0.021,Y -454.132,Z 1087.505,A 0.000,B 0.000,C 90.000,E1 270.917} C_DIS
LIN {X 0.127,Y -447.646,Z 1087.503,A 0.000,B 0.000,C 90.000,E1 270.516} C_DIS
LIN {X -0.176,Y -440.568,Z 1087.501,A 0.000,B 0.000,C 90.000,E1 270.229} C_DIS
LIN {X 0.010,Y -433.076,Z 1087.500,A 0.000,B 0.000,C 90.000,E1 269.943} C_DIS
LIN {X 0.190,Y -425.276,Z 1087.499,A 0.000,B 0.000,C 90.000,E1 269.714} C_DIS
LIN {X -0.126,Y -417.408,Z 1087.498,A 0.000,B 0.000,C 90.000,E1 269.599} C_DIS
LIN {X -0.165,Y -408.736,Z 1087.497,A 0.000,B 0.000,C 90.000,E1 269.484} C_DIS
LIN {X 0.013,Y -397.754,Z 1087.496,A 0.000,B 0.000,C 90.000,E1 269.370} C_DIS
LIN {X -0.116,Y -392.438,Z 1087.496,A 0.000,B 0.000,C 90.000,E1 269.370} C_DIS
LIN {X -0.084,Y -181.399,Z 1087.496,A 0.000,B 0.000,C 90.000,E1 269.370} C_DIS
LIN {X 0.035,Y -180.802,Z 1087.471,A 0.000,B 0.000,C 90.000,E1 264.780} C_DIS
LIN {X -0.068,Y -178.902,Z 1087.443,A 0.000,B 0.000,C 90.000,E1 259.746} C_DIS
LIN {X 0.013,Y -175.945,Z 1087.415,A 0.000,B 0.000,C 90.000,E1 254.629} C_DIS
LIN {X -0.040,Y -175.404,Z 1087.410,A 0.000,B 0.000,C 90.000,E1 253.795} C_DIS
LIN {X -0.036,Y -172.171,Z 1087.386,A 0.000,B 0.000,C 90.000,E1 249.518} C_DIS
LIN {X 0.003,Y -171.641,Z 1087.381,A 0.000,B 0.000,C 90.000,E1 248.646} C_DIS
LIN {X -0.002,Y -167.864,Z 1087.357,A 0.000,B 0.000,C 90.000,E1 244.332} C_DIS
LIN {X -0.060,Y -166.597,Z 1087.348,A 0.000,B 0.000,C 90.000,E1 242.615} C_DIS
LIN {X 0.073,Y -162.586,Z 1087.323,A 0.000,B 0.000,C 90.000,E1 238.201} C_DIS
LIN {X -0.091,Y -161.269,Z 1087.314,A 0.000,B 0.000,C 90.000,E1 236.501} C_DIS
LIN {X 0.042,Y -157.270,Z 1087.289,A 0.000,B 0.000,C 90.000,E1 232.029} C_DIS
LIN {X -0.032,Y -155.990,Z 1087.279,A 0.000,B 0.000,C 90.000,E1 230.275} C_DIS
LIN {X -0.071,Y -152.247,Z 1087.254,A 0.000,B 0.000,C 90.000,E1 225.810} C_DIS
LIN {X -0.048,Y -150.487,Z 1087.239,A 0.000,B 0.000,C 90.000,E1 223.095} C_DIS
LIN {X -0.017,Y -147.211,Z 1087.214,A 0.000,B 0.000,C 90.000,E1 218.543} C_DIS
LIN {X -0.047,Y -145.232,Z 1087.194,A 0.000,B 0.000,C 90.000,E1 214.898} C_DIS
LIN {X 0.064,Y -142.356,Z 1087.163,A 0.000,B 0.000,C 90.000,E1 209.333} C_DIS
LIN {X -0.009,Y -141.743,Z 1087.153,A 0.000,B 0.000,C 90.000,E1 207.513} C_DIS
LIN {X -0.033,Y -139.489,Z 1087.117,A 0.000,B 0.000,C 90.000,E1 201.025} C_DIS
LIN {X -0.047,Y -138.992,Z 1087.101,A 0.000,B 0.000,C 90.000,E1 198.236} C_DIS
LIN {X 0.047,Y -138.335,Z 1087.055,A 0.000,B 0.000,C 90.000,E1 189.792} C_DIS
LIN {X -0.067,Y -139.418,Z 1087.008,A 0.000,B 0.000,C 90.000,E1 181.432} C_DIS
LIN {X -0.015,Y -141.335,Z 1086.972,A 0.000,B 0.000,C 90.000,E1 174.894} C_DIS
LIN {X -0.057,Y -142.691,Z 1086.956,A 0.000,B 0.000,C 90.000,E1 172.129} C_DIS
LIN {X 0.063,Y -145.055,Z 1086.931,A 0.000,B 0.000,C 90.000,E1 167.465} C_DIS
LIN {X 0.060,Y -147.681,Z 1086.910,A 0.000,B 0.000,C 90.000,E1 163.795} C_DIS
LIN {X -0.048,Y -150.326,Z 1086.890,A 0.000,B 0.000,C 90.000,E1 160.188} C_DIS
LIN {X 0.024,Y -153.742,Z 1086.870,A 0.000,B 0.000,C 90.000,E1 156.538} C_DIS
LIN {X 0.015,Y -157.156,Z 1086.850,A 0.000,B 0.000,C 90.000,E1 152.948} C_DIS
LIN {X -0.050,Y -161.307,Z 1086.830,A 0.000,B 0.000,C 90.000,E1 149.410} C_DIS
LIN {X -0.034,Y -164.423,Z 1086.815,A 0.000,B 0.000,C 90.000,E1 146.755} C_DIS
LIN {X -0.037,Y -169.107,Z 1086.796,A 0.000,B 0.000,C 90.000,E1 143.256} C_DIS
LIN {X -0.087,Y -171.661,Z 1086.786,A 0.000,B 0.000,C 90.000,E1 141.537} C_DIS
LIN {X -0.042,Y -176.627,Z 1086.767,A 0.000,B 0.000,C 90.000,E1 138.081} C_DIS
LIN {X 0.086,Y -180.924,Z 1086.753,A 0.000,B 0.000,C 90.000,E1 135.486} C_DIS
LIN {X -0.050,Y -186.342,Z 1086.734,A 0.000,B 0.000,C 90.000,E1 132.162} C_DIS
LIN {X 0.016,Y -190.975,Z 1086.720,A 0.000,B 0.000,C 90.000,E1 129.644} C_DIS
LIN {X -0.065,Y -196.749,Z 1086.702,A 0.000,B 0.000,C 90.000,E1 126.377} C_DIS
LIN {X -0.019,Y -199.659,Z 1086.694,A 0.000,B 0.000,C 90.000,E1 124.898} C_DIS
LIN {X -0.065,Y -307.248,Z 1086.694,A 0.000,B 0.000,C 90.000,E1 124.898} C_DIS
LIN {X -0.054,Y -312.105,Z 1086.693,A 0.000,B 0.000,C 90.000,E1 124.739} C_DIS
LIN {X 0.073,Y -315.276,Z 1086.692,A 0.000,B 0.000,C 90.000,E1 124.485} C_DIS
LIN {X -0.031,Y -318.980,Z 1086.689,A 0.000,B 0.000,C 90.000,E1 124.072} C_DIS
LIN {X -0.185,Y -320.860,Z 1086.688,A 0.000,B 0.000,C 90.000,E1 123.785} C_DIS
LIN {X -0.072,Y -322.330,Z 1086.686,A 0.000,B 0.000,C 90.000,E1 123.452} C_DIS
LIN {X 0.078,Y -335.235,Z 1086.667,A 0.000,B 0.000,C 90.000,E1 119.951} C_DIS
LIN {X -0.001,Y -347.218,Z 1086.651,A 0.000,B 0.000,C 90.000,E1 117.180} C_DIS
LIN {X -0.065,Y -360.666,Z 1086.636,A 0.000,B 0.000,C 90.000,E1 114.463} C_DIS
LIN {X 0.010,Y -373.948,Z 1086.623,A 0.000,B 0.000,C 90.000,E1 112.078} C_DIS
LIN {X -0.003,Y -388.577,Z 1086.610,A 0.000,B 0.000,C 90.000,E1 109.758} C_DIS
LIN {X -0.155,Y -404.654,Z 1086.597,A 0.000,B 0.000,C 90.000,E1 107.511} C_DIS
LIN {X 0.238,Y -422.295,Z 1086.585,A 0.000,B 0.000,C 90.000,E1 105.245} C_DIS
LIN {X 0.083,Y -441.571,Z 1086.573,A 0.000,B 0.000,C 90.000,E1 103.119} C_DIS
LIN {X -0.001,Y -461.737,Z 1086.562,A 0.000,B 0.000,C 90.000,E1 101.130} C_DIS
LIN {X -0.018,Y -466.863,Z 1086.559,A 0.000,B 0.000,C 90.000,E1 100.658} C_DIS
LIN {X -0.007,Y -469.182,Z 1086.558,A 0.000,B 0.000,C 90.000,E1 100.423} C_DIS
LIN {X -0.203,Y -471.025,Z 1086.557,A 0.000,B 0.000,C 90.000,E1 100.197} C_DIS
LIN {X 0.149,Y -472.415,Z 1086.555,A 0.000,B 0.000,C 90.000,E1 99.905} C_DIS
LIN {X -0.137,Y -474.216,Z 1086.552,A 0.000,B 0.000,C 90.000,E1 99.434} C_DIS
LIN {X -0.026,Y -474.928,Z 1086.550,A 0.000,B 0.000,C 90.000,E1 98.916} C_DIS
LIN {X 0.099,Y -474.670,Z 1086.547,A 0.000,B 0.000,C 90.000,E1 98.398} C_DIS
LIN {X -0.240,Y -473.408,Z 1086.544,A 0.000,B 0.000,C 90.000,E1 97.936} C_DIS
LIN {X 0.091,Y -472.340,Z 1086.542,A 0.000,B 0.000,C 90.000,E1 97.644} C_DIS
LIN {X -0.048,Y -470.912,Z 1086.541,A 0.000,B 0.000,C 90.000,E1 97.409} C_DIS
LIN {X -0.170,Y -456.608,Z 1086.530,A 0.000,B 0.000,C 90.000,E1 95.391} C_DIS
LIN {X -0.027,Y -440.594,Z 1086.517,A 0.000,B 0.000,C 90.000,E1 93.037} C_DIS
LIN {X 0.106,Y -425.991,Z 1086.504,A 0.000,B 0.000,C 90.000,E1 90.630} C_DIS
LIN {X 0.037,Y -409.301,Z 1086.487,A 0.000,B 0.000,C 90.000,E1 87.650} C_DIS
LIN {X 0.038,Y -400.391,Z 1086.478,A 0.000,B 0.000,C 90.000,E1 85.988} C_DIS
LIN {X -0.063,Y -391.226,Z 1086.468,A 0.000,B 0.000,C 90.000,E1 84.318} C_DIS
LIN {X 0.093,Y -380.476,Z 1086.457,A 0.000,B 0.000,C 90.000,E1 82.299} C_DIS
LIN {X 0.118,Y -372.673,Z 1086.449,A 0.000,B 0.000,C 90.000,E1 80.849} C_DIS
LIN {X 0.009,Y -362.970,Z 1086.439,A 0.000,B 0.000,C 90.000,E1 79.106} C_DIS
LIN {X 0.139,Y -353.035,Z 1086.430,A 0.000,B 0.000,C 90.000,E1 77.297} C_DIS
LIN {X -0.176,Y -341.394,Z 1086.418,A 0.000,B 0.000,C 90.000,E1 75.227} C_DIS
LIN {X -0.189,Y -325.240,Z 1086.401,A 0.000,B 0.000,C 90.000,E1 72.127} C_DIS
LIN {X -0.073,Y -308.569,Z 1086.381,A 0.000,B 0.000,C 90.000,E1 68.592} C_DIS
LIN {X -0.076,Y -297.145,Z 1086.366,A 0.000,B 0.000,C 90.000,E1 65.973} C_DIS
LIN {X 0.144,Y -285.948,Z 1086.352,A 0.000,B 0.000,C 90.000,E1 63.256} C_DIS
LIN {X -0.114,Y -276.364,Z 1086.338,A 0.000,B 0.000,C 90.000,E1 60.923} C_DIS
LIN {X -0.008,Y -265.703,Z 1086.323,A 0.000,B 0.000,C 90.000,E1 58.122} C_DIS
LIN {X 0.104,Y -255.407,Z 1086.307,A 0.000,B 0.000,C 90.000,E1 55.261} C_DIS
LIN {X -0.016,Y -244.360,Z 1086.289,A 0.000,B 0.000,C 90.000,E1 52.029} C_DIS
LIN {X 0.026,Y -234.059,Z 1086.271,A 0.000,B 0.000,C 90.000,E1 48.690} C_DIS
LIN {X 0.013,Y -223.486,Z 1086.250,A 0.000,B 0.000,C 90.000,E1 44.919} C_DIS
LIN {X 0.025,Y -215.428,Z 1086.232,A 0.000,B 0.000,C 90.000,E1 41.838} C_DIS
LIN {X 0.036,Y -207.744,Z 1086.215,A 0.000,B 0.000,C 90.000,E1 38.705} C_DIS
LIN {X 0.051,Y -200.611,Z 1086.197,A 0.000,B 0.000,C 90.000,E1 35.518} C_DIS
LIN {X 0.033,Y -194.068,Z 1086.179,A 0.000,B 0.000,C 90.000,E1 32.291} C_DIS
LIN {X -0.014,Y -188.205,Z 1086.161,A 0.000,B 0.000,C 90.000,E1 29.027} C_DIS
LIN {X -0.058,Y -183.116,Z 1086.143,A 0.000,B 0.000,C 90.000,E1 25.720} C_DIS
LIN {X 0.028,Y -178.721,Z 1086.124,A 0.000,B 0.000,C 90.000,E1 22.333} C_DIS
LIN {X -0.037,Y -174.134,Z 1086.101,A 0.000,B 0.000,C 90.000,E1 18.109} C_DIS
LIN {X -0.059,Y -170.668,Z 1086.077,A 0.000,B 0.000,C 90.000,E1 13.828} C_DIS
LIN {X -0.015,Y -167.848,Z 1086.048,A 0.000,B 0.000,C 90.000,E1 8.624} C_DIS
LIN {X 0.081,Y -168.585,Z 1085.949,A 0.000,B 0.000,C 90.000,E1 350.792} C_DIS
LIN {X 0.068,Y -171.301,Z 1085.925,A 0.000,B 0.000,C 90.000,E1 346.464} C_DIS
LIN {X 0.009,Y -175.054,Z 1085.901,A 0.000,B 0.000,C 90.000,E1 342.181} C_DIS
LIN {X -0.011,Y -178.832,Z 1085.882,A 0.000,B 0.000,C 90.000,E1 338.773} C_DIS
LIN {X 0.093,Y -183.242,Z 1085.863,A 0.000,B 0.000,C 90.000,E1 335.357} C_DIS
LIN {X 0.038,Y -188.368,Z 1085.845,A 0.000,B 0.000,C 90.000,E1 332.025} C_DIS
LIN {X -0.047,Y -194.350,Z 1085.826,A 0.000,B 0.000,C 90.000,E1 328.742} C_DIS
LIN {X -0.017,Y -201.102,Z 1085.808,A 0.000,B 0.000,C 90.000,E1 325.468} C_DIS
LIN {X -0.086,Y -208.578,Z 1085.790,A 0.000,B 0.000,C 90.000,E1 322.271} C_DIS
LIN {X -0.026,Y -216.708,Z 1085.773,A 0.000,B 0.000,C 90.000,E1 319.094} C_DIS
LIN {X 0.055,Y -225.714,Z 1085.755,A 0.000,B 0.000,C 90.000,E1 315.972} C_DIS
LIN {X 0.049,Y -235.765,Z 1085.739,A 0.000,B 0.000,C 90.000,E1 312.933} C_DIS
LIN {X 0.012,Y -245.716,Z 1085.724,A 0.000,B 0.000,C 90.000,E1 310.334} C_DIS
LIN {X -0.131,Y -257.101,Z 1085.710,A 0.000,B 0.000,C 90.000,E1 307.810} C_DIS
LIN {X -0.038,Y -267.743,Z 1085.698,A 0.000,B 0.000,C 90.000,E1 305.644} C_DIS
LIN {X 0.027,Y -285.102,Z 1085.681,A 0.000,B 0.000,C 90.000,E1 302.498} C_DIS
LIN {X 0.055,Y -303.939,Z 1085.664,A 0.000,B 0.000,C 90.000,E1 299.461} C_DIS
LIN {X 0.025,Y -324.435,Z 1085.647,A 0.000,B 0.000,C 90.000,E1 296.539} C_DIS
LIN {X 0.063,Y -336.750,Z 1085.639,A 0.000,B 0.000,C 90.000,E1 294.951} C_DIS
LIN {X -0.166,Y -352.296,Z 1085.629,A 0.000,B 0.000,C 90.000,E1 293.206} C_DIS
LIN {X 0.023,Y -365.162,Z 1085.621,A 0.000,B 0.000,C 90.000,E1 291.844} C_DIS
LIN {X -0.076,Y -384.612,Z 1085.611,A 0.000,B 0.000,C 90.000,E1 290.066} C_DIS
LIN {X -0.057,Y -401.054,Z 1085.604,A 0.000,B 0.000,C 90.000,E1 288.652} C_DIS
LIN {X 0.002,Y -414.596,Z 1085.597,A 0.000,B 0.000,C 90.000,E1 287.457} C_DIS
LIN {X 0.044,Y -422.407,Z 1085.593,A 0.000,B 0.000,C 90.000,E1 286.732} C_DIS
LIN {X 0.061,Y -432.531,Z 1085.587,A 0.000,B 0.000,C 90.000,E1 285.733} C_DIS
LIN {X 0.058,Y -439.905,Z 1085.583,A 0.000,B 0.000,C 90.000,E1 284.954} C_DIS
LIN {X -0.045,Y -446.925,Z 1085.579,A 0.000,B 0.000,C 90.000,E1 284.175} C_DIS
LIN {X 0.225,Y -453.370,Z 1085.574,A 0.000,B 0.000,C 90.000,E1 283.355} C_DIS
LIN {X 0.112,Y -459.211,Z 1085.570,A 0.000,B 0.000,C 90.000,E1 282.591} C_DIS
LIN {X 0.052,Y -464.312,Z 1085.566,A 0.000,B 0.000,C 90.000,E1 281.827} C_DIS
LIN {X 0.188,Y -467.310,Z 1085.563,A 0.000,B 0.000,C 90.000,E1 281.299} C_DIS
LIN {X 0.103,Y -471.113,Z 1085.559,A 0.000,B 0.000,C 90.000,E1 280.546} C_DIS
LIN {X -0.186,Y -473.308,Z 1085.556,A 0.000,B 0.000,C 90.000,E1 280.074} C_DIS
LIN {X -0.079,Y -475.235,Z 1085.553,A 0.000,B 0.000,C 90.000,E1 279.557} C_DIS
LIN {X 0.115,Y -476.899,Z 1085.550,A 0.000,B 0.000,C 90.000,E1 279.029} C_DIS
LIN {X -0.228,Y -478.332,Z 1085.547,A 0.000,B 0.000,C 90.000,E1 278.568} C_DIS
LIN {X -0.086,Y -479.553,Z 1085.545,A 0.000,B 0.000,C 90.000,E1 278.049} C_DIS
LIN {X 0.066,Y -480.584,Z 1085.542,A 0.000,B 0.000,C 90.000,E1 277.530} C_DIS
LIN {X -0.250,Y -481.417,Z 1085.539,A 0.000,B 0.000,C 90.000,E1 277.068} C_DIS
LIN {X -0.082,Y -482.027,Z 1085.536,A 0.000,B 0.000,C 90.000,E1 276.549} C_DIS
LIN {X 0.091,Y -482.404,Z 1085.534,A 0.000,B 0.000,C 90.000,E1 276.030} C_DIS
LIN {X -0.212,Y -482.445,Z 1085.531,A 0.000,B 0.000,C 90.000,E1 275.568} C_DIS
LIN {X -0.035,Y -482.058,Z 1085.528,A 0.000,B 0.000,C 90.000,E1 275.049} C_DIS
LIN {X 0.140,Y -481.260,Z 1085.525,A 0.000,B 0.000,C 90.000,E1 274.531} C_DIS
LIN {X -0.169,Y -479.993,Z 1085.522,A 0.000,B 0.000,C 90.000,E1 274.069} C_DIS
LIN {X -0.036,Y -478.158,Z 1085.520,A 0.000,B 0.000,C 90.000,E1 273.555} C_DIS
LIN {X 0.118,Y -475.651,Z 1085.517,A 0.000,B 0.000,C 90.000,E1 273.037} C_DIS
LIN {X 0.228,Y -472.374,Z 1085.514,A 0.000,B 0.000,C 90.000,E1 272.522} C_DIS
LIN {X -0.145,Y -468.227,Z 1085.511,A 0.000,B 0.000,C 90.000,E1 272.064} C_DIS
LIN {X 0.142,Y -465.743,Z 1085.510,A 0.000,B 0.000,C 90.000,E1 271.776} C_DIS
LIN {X -0.089,Y -460.133,Z 1085.507,A 0.000,B 0.000,C 90.000,E1 271.318} C_DIS
LIN {X 0.071,Y -453.946,Z 1085.505,A 0.000,B 0.000,C 90.000,E1 270.859} C_DIS
LIN {X -0.222,Y -447.349,Z 1085.503,A 0.000,B 0.000,C 90.000,E1 270.516} C_DIS
LIN {X -0.043,Y -440.298,Z 1085.501,A 0.000,B 0.000,C 90.000,E1 270.172} C_DIS
LIN {X 0.176,Y -432.713,Z 1085.500,A 0.000,B 0.000,C 90.000,E1 269.885} C_DIS
LIN {X -0.026,Y -424.945,Z 1085.498,A 0.000,B 0.000,C 90.000,E1 269.714} C_DIS
LIN {X 0.103,Y -416.980,Z 1085.498,A 0.000,B 0.000,C 90.000,E1 269.542} C_DIS
LIN {X 0.064,Y -408.008,Z 1085.497,A 0.000,B 0.000,C 90.000,E1 269.427} C_DIS
LIN {X -0.145,Y -395.595,Z 1085.496,A 0.000,B 0.000,C 90.000,E1 269.370} C_DIS
LIN {X 0.186,Y -390.436,Z 1085.496,A 0.000,B 0.000,C 90.000,E1 269.312} C_DIS
LIN {X 0.058,Y -181.396,Z 1085.496,A 0.000,B 0.000,C 90.000,E1 269.312} C_DIS
LIN {X -0.031,Y -180.794,Z 1085.471,A 0.000,B 0.000,C 90.000,E1 264.780} C_DIS
LIN {X 0.043,Y -178.893,Z 1085.443,A 0.000,B 0.000,C 90.000,E1 259.690} C_DIS
LIN {X -0.053,Y -175.936,Z 1085.415,A 0.000,B 0.000,C 90.000,E1 254.629} C_DIS
LIN {X 0.063,Y -175.386,Z 1085.410,A 0.000,B 0.000,C 90.000,E1 253.740} C_DIS
LIN {X -0.102,Y -172.157,Z 1085.386,A 0.000,B 0.000,C 90.000,E1 249.518} C_DIS
LIN {X -0.063,Y -171.625,Z 1085.381,A 0.000,B 0.000,C 90.000,E1 248.646} C_DIS
LIN {X 0.085,Y -167.848,Z 1085.357,A 0.000,B 0.000,C 90.000,E1 244.280} C_DIS
LIN {X 0.025,Y -166.577,Z 1085.348,A 0.000,B 0.000,C 90.000,E1 242.564} C_DIS
LIN {X 0.011,Y -162.569,Z 1085.323,A 0.000,B 0.000,C 90.000,E1 238.201} C_DIS
LIN {X 0.071,Y -161.250,Z 1085.314,A 0.000,B 0.000,C 90.000,E1 236.421} C_DIS
LIN {X -0.019,Y -157.253,Z 1085.289,A 0.000,B 0.000,C 90.000,E1 232.029} C_DIS
LIN {X 0.028,Y -155.975,Z 1085.279,A 0.000,B 0.000,C 90.000,E1 230.231} C_DIS
LIN {X 0.084,Y -152.230,Z 1085.254,A 0.000,B 0.000,C 90.000,E1 225.729} C_DIS
LIN {X -0.005,Y -150.472,Z 1085.239,A 0.000,B 0.000,C 90.000,E1 223.056} C_DIS
LIN {X -0.077,Y -147.197,Z 1085.214,A 0.000,B 0.000,C 90.000,E1 218.543} C_DIS
LIN {X -0.023,Y -145.216,Z 1085.194,A 0.000,B 0.000,C 90.000,E1 214.865} C_DIS
LIN {X 0.005,Y -142.347,Z 1085.163,A 0.000,B 0.000,C 90.000,E1 209.333} C_DIS
LIN {X -0.067,Y -141.734,Z 1085.153,A 0.000,B 0.000,C 90.000,E1 207.513} C_DIS
LIN {X 0.040,Y -139.484,Z 1085.117,A 0.000,B 0.000,C 90.000,E1 200.972} C_DIS
LIN {X 0.030,Y -138.985,Z 1085.101,A 0.000,B 0.000,C 90.000,E1 198.181} C_DIS
LIN {X -0.009,Y -138.334,Z 1085.054,A 0.000,B 0.000,C 90.000,E1 189.792} C_DIS
LIN {X 0.015,Y -139.423,Z 1085.008,A 0.000,B 0.000,C 90.000,E1 181.375} C_DIS
LIN {X 0.069,Y -141.345,Z 1084.971,A 0.000,B 0.000,C 90.000,E1 174.837} C_DIS
LIN {X 0.046,Y -142.701,Z 1084.956,A 0.000,B 0.000,C 90.000,E1 172.064} C_DIS
LIN {X 0.005,Y -145.070,Z 1084.930,A 0.000,B 0.000,C 90.000,E1 167.465} C_DIS
LIN {X 0.001,Y -147.695,Z 1084.910,A 0.000,B 0.000,C 90.000,E1 163.795} C_DIS
LIN {X 0.034,Y -150.345,Z 1084.890,A 0.000,B 0.000,C 90.000,E1 160.134} C_DIS
LIN {X 0.027,Y -154.600,Z 1084.865,A 0.000,B 0.000,C 90.000,E1 155.613} C_DIS
LIN {X 0.035,Y -158.140,Z 1084.845,A 0.000,B 0.000,C 90.000,E1 152.025} C_DIS
LIN {X 0.080,Y -162.426,Z 1084.825,A 0.000,B 0.000,C 90.000,E1 148.456} C_DIS
LIN {X -0.024,Y -166.684,Z 1084.805,A 0.000,B 0.000,C 90.000,E1 144.975} C_DIS
LIN {X 0.089,Y -171.690,Z 1084.786,A 0.000,B 0.000,C 90.000,E1 141.457} C_DIS
LIN {X 0.023,Y -176.661,Z 1084.767,A 0.000,B 0.000,C 90.000,E1 138.038} C_DIS
LIN {X 0.019,Y -180.957,Z 1084.753,A 0.000,B 0.000,C 90.000,E1 135.486} C_DIS
LIN {X 0.007,Y -186.380,Z 1084.734,A 0.000,B 0.000,C 90.000,E1 132.123} C_DIS
LIN {X -0.053,Y -191.010,Z 1084.720,A 0.000,B 0.000,C 90.000,E1 129.644} C_DIS
LIN {X -0.019,Y -196.789,Z 1084.702,A 0.000,B 0.000,C 90.000,E1 126.343} C_DIS
LIN {X -0.038,Y -199.573,Z 1084.694,A 0.000,B 0.000,C 90.000,E1 124.945} C_DIS
LIN {X -0.094,Y -306.502,Z 1084.694,A 0.000,B 0.000,C 90.000,E1 124.945} C_DIS
LIN {X 0.047,Y -308.198,Z 1084.694,A 0.000,B 0.000,C 90.000,E1 124.898} C_DIS
LIN {X 0.092,Y -312.907,Z 1084.693,A 0.000,B 0.000,C 90.000,E1 124.692} C_DIS
LIN {X -0.040,Y -316.061,Z 1084.691,A 0.000,B 0.000,C 90.000,E1 124.452} C_DIS
LIN {X -0.180,Y -319.752,Z 1084.689,A 0.000,B 0.000,C 90.000,E1 123.992} C_DIS
LIN {X 0.066,Y -321.465,Z 1084.687,A 0.000,B 0.000,C 90.000,E1 123.627} C_DIS
LIN {X -0.050,Y -323.911,Z 1084.683,A 0.000,B 0.000,C 90.000,E1 123.007} C_DIS
LIN {X 0.167,Y -334.442,Z 1084.667,A 0.000,B 0.000,C 90.000,E1 120.129} C_DIS
LIN {X -0.095,Y -346.327,Z 1084.652,A 0.000,B 0.000,C 90.000,E1 117.385} C_DIS
LIN {X -0.037,Y -359.674,Z 1084.637,A 0.000,B 0.000,C 90.000,E1 114.643} C_DIS
LIN {X -0.131,Y -372.856,Z 1084.624,A 0.000,B 0.000,C 90.000,E1 112.280} C_DIS
LIN {X -0.034,Y -387.378,Z 1084.611,A 0.000,B 0.000,C 90.000,E1 109.939} C_DIS
LIN {X 0.167,Y -403.339,Z 1084.598,A 0.000,B 0.000,C 90.000,E1 107.638} C_DIS
LIN {X 0.140,Y -420.856,Z 1084.586,A 0.000,B 0.000,C 90.000,E1 105.426} C_DIS
LIN {X -0.074,Y -440.026,Z 1084.574,A 0.000,B 0.000,C 90.000,E1 103.300} C_DIS
LIN {X -0.176,Y -460.148,Z 1084.563,A 0.000,B 0.000,C 90.000,E1 101.299} C_DIS
LIN {X 0.168,Y -467.802,Z 1084.559,A 0.000,B 0.000,C 90.000,E1 100.546} C_DIS
LIN {X 0.189,Y -469.871,Z 1084.557,A 0.000,B 0.000,C 90.000,E1 100.310} C_DIS
LIN {X 0.038,Y -471.563,Z 1084.556,A 0.000,B 0.000,C 90.000,E1 100.074} C_DIS
LIN {X -0.194,Y -472.834,Z 1084.555,A 0.000,B 0.000,C 90.000,E1 99.849} C_DIS
LIN {X -0.011,Y -474.404,Z 1084.552,A 0.000,B 0.000,C 90.000,E1 99.321} C_DIS
LIN {X 0.105,Y -474.923,Z 1084.549,A 0.000,B 0.000,C 90.000,E1 98.803} C_DIS
LIN {X -0.237,Y -474.479,Z 1084.546,A 0.000,B 0.000,C 90.000,E1 98.341} C_DIS
LIN {X -0.041,Y -473.007,Z 1084.543,A 0.000,B 0.000,C 90.000,E1 97.814} C_DIS
LIN {X -0.242,Y -471.809,Z 1084.542,A 0.000,B 0.000,C 90.000,E1 97.587} C_DIS
LIN {X -0.121,Y -468.386,Z 1084.539,A 0.000,B 0.000,C 90.000,E1 97.068} C_DIS
LIN {X -0.052,Y -455.899,Z 1084.529,A 0.000,B 0.000,C 90.000,E1 95.277} C_DIS
LIN {X -0.132,Y -441.605,Z 1084.518,A 0.000,B 0.000,C 90.000,E1 93.212} C_DIS
LIN {X 0.048,Y -426.974,Z 1084.505,A 0.000,B 0.000,C 90.000,E1 90.802} C_DIS
LIN {X -0.072,Y -411.654,Z 1084.489,A 0.000,B 0.000,C 90.000,E1 88.108} C_DIS
LIN {X -0.021,Y -402.808,Z 1084.480,A 0.000,B 0.000,C 90.000,E1 86.445} C_DIS
LIN {X -0.108,Y -393.696,Z 1084.471,A 0.000,B 0.000,C 90.000,E1 84.780} C_DIS
LIN {X 0.128,Y -381.397,Z 1084.458,A 0.000,B 0.000,C 90.000,E1 82.470} C_DIS
LIN {X 0.119,Y -372.034,Z 1084.449,A 0.000,B 0.000,C 90.000,E1 80.735} C_DIS
LIN {X -0.005,Y -362.287,Z 1084.439,A 0.000,B 0.000,C 90.000,E1 78.993} C_DIS
LIN {X -0.158,Y -352.355,Z 1084.429,A 0.000,B 0.000,C 90.000,E1 77.229} C_DIS
LIN {X -0.137,Y -340.711,Z 1084.417,A 0.000,B 0.000,C 90.000,E1 75.102} C_DIS
LIN {X 0.143,Y -324.581,Z 1084.400,A 0.000,B 0.000,C 90.000,E1 71.945} C_DIS
LIN {X -0.066,Y -307.964,Z 1084.380,A 0.000,B 0.000,C 90.000,E1 68.465} C_DIS
LIN {X -0.085,Y -297.950,Z 1084.368,A 0.000,B 0.000,C 90.000,E1 66.177} C_DIS
LIN {X -0.107,Y -286.733,Z 1084.353,A 0.000,B 0.000,C 90.000,E1 63.512} C_DIS
LIN {X -0.102,Y -277.111,Z 1084.339,A 0.000,B 0.000,C 90.000,E1 61.129} C_DIS
LIN {X 0.019,Y -266.406,Z 1084.324,A 0.000,B 0.000,C 90.000,E1 58.329} C_DIS
LIN {X -0.064,Y -256.075,Z 1084.308,A 0.000,B 0.000,C 90.000,E1 55.515} C_DIS
LIN {X -0.101,Y -244.985,Z 1084.290,A 0.000,B 0.000,C 90.000,E1 52.271} C_DIS
LIN {X -0.049,Y -234.612,Z 1084.272,A 0.000,B 0.000,C 90.000,E1 48.933} C_DIS
LIN {X 0.011,Y -224.966,Z 1084.253,A 0.000,B 0.000,C 90.000,E1 45.526} C_DIS
LIN {X 0.053,Y -216.819,Z 1084.236,A 0.000,B 0.000,C 90.000,E1 42.447} C_DIS
LIN {X -0.066,Y -209.019,Z 1084.219,A 0.000,B 0.000,C 90.000,E1 39.358} C_DIS
LIN {X -0.015,Y -201.746,Z 1084.201,A 0.000,B 0.000,C 90.000,E1 36.171} C_DIS
LIN {X -0.054,Y -195.097,Z 1084.183,A 0.000,B 0.000,C 90.000,E1 32.959} C_DIS
LIN {X 0.018,Y -189.054,Z 1084.165,A 0.000,B 0.000,C 90.000,E1 29.667} C_DIS
LIN {X -0.009,Y -183.831,Z 1084.146,A 0.000,B 0.000,C 90.000,E1 26.360} C_DIS
LIN {X -0.069,Y -179.291,Z 1084.128,A 0.000,B 0.000,C 90.000,E1 23.025} C_DIS
LIN {X -0.048,Y -174.555,Z 1084.104,A 0.000,B 0.000,C 90.000,E1 18.779} C_DIS
LIN {X -0.008,Y -170.915,Z 1084.080,A 0.000,B 0.000,C 90.000,E1 14.481} C_DIS
LIN {X 0.080,Y -167.920,Z 1084.052,A 0.000,B 0.000,C 90.000,E1 9.265} C_DIS
LIN {X 0.069,Y -166.045,Z 1084.008,A 0.000,B 0.000,C 90.000,E1 1.432} C_DIS
LIN {X 0.060,Y -167.623,Z 1083.959,A 0.000,B 0.000,C 90.000,E1 352.534} C_DIS
LIN {X -0.055,Y -169.880,Z 1083.934,A 0.000,B 0.000,C 90.000,E1 348.229} C_DIS
LIN {X -0.084,Y -173.198,Z 1083.911,A 0.000,B 0.000,C 90.000,E1 343.921} C_DIS
LIN {X -0.044,Y -177.620,Z 1083.887,A 0.000,B 0.000,C 90.000,E1 339.625} C_DIS
LIN {X -0.039,Y -181.873,Z 1083.868,A 0.000,B 0.000,C 90.000,E1 336.230} C_DIS
LIN {X -0.044,Y -186.814,Z 1083.849,A 0.000,B 0.000,C 90.000,E1 332.871} C_DIS
LIN {X -0.003,Y -192.573,Z 1083.831,A 0.000,B 0.000,C 90.000,E1 329.537} C_DIS
LIN {X -0.123,Y -199.195,Z 1083.813,A 0.000,B 0.000,C 90.000,E1 326.294} C_DIS
LIN {X -0.074,Y -206.504,Z 1083.795,A 0.000,B 0.000,C 90.000,E1 323.050} C_DIS
LIN {X 0.001,Y -215.515,Z 1083.775,A 0.000,B 0.000,C 90.000,E1 319.461} C_DIS
LIN {X -0.098,Y -224.425,Z 1083.758,A 0.000,B 0.000,C 90.000,E1 316.377} C_DIS
LIN {X 0.017,Y -234.301,Z 1083.741,A 0.000,B 0.000,C 90.000,E1 313.299} C_DIS
LIN {X -0.065,Y -244.051,Z 1083.726,A 0.000,B 0.000,C 90.000,E1 310.701} C_DIS
LIN {X 0.115,Y -255.283,Z 1083.712,A 0.000,B 0.000,C 90.000,E1 308.096} C_DIS
LIN {X 0.025,Y -265.785,Z 1083.700,A 0.000,B 0.000,C 90.000,E1 305.964} C_DIS
LIN {X -0.041,Y -283.007,Z 1083.682,A 0.000,B 0.000,C 90.000,E1 302.832} C_DIS
LIN {X -0.073,Y -301.752,Z 1083.665,A 0.000,B 0.000,C 90.000,E1 299.795} C_DIS
LIN {X -0.094,Y -319.744,Z 1083.651,A 0.000,B 0.000,C 90.000,E1 297.180} C_DIS
LIN {X -0.174,Y -334.241,Z 1083.640,A 0.000,B 0.000,C 90.000,E1 295.283} C_DIS
LIN {X -0.112,Y -349.759,Z 1083.630,A 0.000,B 0.000,C 90.000,E1 293.462} C_DIS
LIN {X 0.062,Y -363.213,Z 1083.622,A 0.000,B 0.000,C 90.000,E1 292.025} C_DIS
LIN {X -0.023,Y -382.433,Z 1083.612,A 0.000,B 0.000,C 90.000,E1 290.248} C_DIS
LIN {X -0.093,Y -401.745,Z 1083.603,A 0.000,B 0.000,C 90.000,E1 288.598} C_DIS
LIN {X -0.003,Y -415.224,Z 1083.597,A 0.000,B 0.000,C 90.000,E1 287.402} C_DIS
LIN {X 0.003,Y -423.056,Z 1083.593,A 0.000,B 0.000,C 90.000,E1 286.677} C_DIS
LIN {X 0.249,Y -430.695,Z 1083.589,A 0.000,B 0.000,C 90.000,E1 285.898} C_DIS
LIN {X 0.179,Y -438.104,Z 1083.584,A 0.000,B 0.000,C 90.000,E1 285.134} C_DIS
LIN {X 0.051,Y -445.290,Z 1083.580,A 0.000,B 0.000,C 90.000,E1 284.356} C_DIS
LIN {X -0.137,Y -451.865,Z 1083.575,A 0.000,B 0.000,C 90.000,E1 283.592} C_DIS
LIN {X 0.184,Y -457.888,Z 1083.571,A 0.000,B 0.000,C 90.000,E1 282.771} C_DIS
LIN {X 0.112,Y -463.224,Z 1083.567,A 0.000,B 0.000,C 90.000,E1 282.007} C_DIS
LIN {X 0.087,Y -467.750,Z 1083.563,A 0.000,B 0.000,C 90.000,E1 281.243} C_DIS
LIN {X 0.007,Y -471.502,Z 1083.558,A 0.000,B 0.000,C 90.000,E1 280.489} C_DIS
LIN {X 0.186,Y -473.669,Z 1083.555,A 0.000,B 0.000,C 90.000,E1 279.962} C_DIS
LIN {X -0.169,Y -475.571,Z 1083.553,A 0.000,B 0.000,C 90.000,E1 279.500} C_DIS
LIN {X 0.026,Y -477.237,Z 1083.550,A 0.000,B 0.000,C 90.000,E1 278.973} C_DIS
LIN {X -0.170,Y -479.880,Z 1083.544,A 0.000,B 0.000,C 90.000,E1 277.992} C_DIS
LIN {X 0.047,Y -480.903,Z 1083.542,A 0.000,B 0.000,C 90.000,E1 277.466} C_DIS
LIN {X 0.207,Y -481.714,Z 1083.539,A 0.000,B 0.000,C 90.000,E1 276.947} C_DIS
LIN {X -0.105,Y -482.311,Z 1083.536,A 0.000,B 0.000,C 90.000,E1 276.486} C_DIS
LIN {X 0.066,Y -482.683,Z 1083.533,A 0.000,B 0.000,C 90.000,E1 275.967} C_DIS
LIN {X 0.195,Y -482.695,Z 1083.530,A 0.000,B 0.000,C 90.000,E1 275.454} C_DIS
LIN {X -0.106,Y -482.289,Z 1083.528,A 0.000,B 0.000,C 90.000,E1 274.992} C_DIS
LIN {X 0.071,Y -481.441,Z 1083.525,A 0.000,B 0.000,C 90.000,E1 274.473} C_DIS
LIN {X 0.242,Y -480.092,Z 1083.522,A 0.000,B 0.000,C 90.000,E1 273.955} C_DIS
LIN {X -0.102,Y -478.211,Z 1083.519,A 0.000,B 0.000,C 90.000,E1 273.498} C_DIS
LIN {X 0.053,Y -475.614,Z 1083.517,A 0.000,B 0.000,C 90.000,E1 272.980} C_DIS
LIN {X 0.164,Y -472.253,Z 1083.514,A 0.000,B 0.000,C 90.000,E1 272.465} C_DIS
LIN {X -0.208,Y -467.972,Z 1083.511,A 0.000,B 0.000,C 90.000,E1 272.007} C_DIS
LIN {X -0.118,Y -462.602,Z 1083.508,A 0.000,B 0.000,C 90.000,E1 271.489} C_DIS
LIN {X -0.155,Y -456.574,Z 1083.506,A 0.000,B 0.000,C 90.000,E1 271.031} C_DIS
LIN {X -0.207,Y -450.066,Z 1083.503,A 0.000,B 0.000,C 90.000,E1 270.630} C_DIS
LIN {X -0.194,Y -443.196,Z 1083.501,A 0.000,B 0.000,C 90.000,E1 270.286} C_DIS
LIN {X -0.143,Y -435.964,Z 1083.500,A 0.000,B 0.000,C 90.000,E1 270.000} C_DIS
LIN {X -0.105,Y -427.936,Z 1083.499,A 0.000,B 0.000,C 90.000,E1 269.771} C_DIS
LIN {X -0.064,Y -420.047,Z 1083.498,A 0.000,B 0.000,C 90.000,E1 269.599} C_DIS
LIN {X -0.144,Y -411.879,Z 1083.497,A 0.000,B 0.000,C 90.000,E1 269.484} C_DIS
LIN {X -0.136,Y -398.952,Z 1083.496,A 0.000,B 0.000,C 90.000,E1 269.370} C_DIS
LIN {X 0.138,Y -393.990,Z 1083.496,A 0.000,B 0.000,C 90.000,E1 269.312} C_DIS
LIN {X 0.036,Y -181.395,Z 1083.496,A 0.000,B 0.000,C 90.000,E1 269.312} C_DIS
LIN {X -0.081,Y -180.788,Z 1083.471,A 0.000,B 0.000,C 90.000,E1 264.780} C_DIS
LIN {X -0.007,Y -178.887,Z 1083.443,A 0.000,B 0.000,C 90.000,E1 259.690} C_DIS
LIN {X 0.068,Y -175.929,Z 1083.414,A 0.000,B 0.000,C 90.000,E1 254.574} C_DIS
LIN {X 0.013,Y -175.371,Z 1083.410,A 0.000,B 0.000,C 90.000,E1 253.740} C_DIS
LIN {X 0.072,Y -172.148,Z 1083.386,A 0.000,B 0.000,C 90.000,E1 249.444} C_DIS
LIN {X 0.050,Y -171.613,Z 1083.381,A 0.000,B 0.000,C 90.000,E1 248.592} C_DIS
LIN {X 0.038,Y -167.835,Z 1083.357,A 0.000,B 0.000,C 90.000,E1 244.280} C_DIS
LIN {X 0.054,Y -166.562,Z 1083.348,A 0.000,B 0.000,C 90.000,E1 242.538} C_DIS
LIN {X -0.036,Y -162.556,Z 1083.323,A 0.000,B 0.000,C 90.000,E1 238.201} C_DIS
LIN {X 0.025,Y -161.235,Z 1083.313,A 0.000,B 0.000,C 90.000,E1 236.421} C_DIS
LIN {X 0.059,Y -157.240,Z 1083.289,A 0.000,B 0.000,C 90.000,E1 231.984} C_DIS
LIN {X -0.018,Y -155.964,Z 1083.279,A 0.000,B 0.000,C 90.000,E1 230.231} C_DIS
LIN {X 0.040,Y -152.218,Z 1083.254,A 0.000,B 0.000,C 90.000,E1 225.729} C_DIS
LIN {X 0.061,Y -150.462,Z 1083.239,A 0.000,B 0.000,C 90.000,E1 223.014} C_DIS
LIN {X 0.086,Y -147.187,Z 1083.214,A 0.000,B 0.000,C 90.000,E1 218.463} C_DIS
LIN {X 0.053,Y -145.205,Z 1083.194,A 0.000,B 0.000,C 90.000,E1 214.818} C_DIS
LIN {X -0.037,Y -142.341,Z 1083.163,A 0.000,B 0.000,C 90.000,E1 209.333} C_DIS
LIN {X 0.016,Y -141.729,Z 1083.153,A 0.000,B 0.000,C 90.000,E1 207.462} C_DIS
LIN {X -0.001,Y -139.481,Z 1083.116,A 0.000,B 0.000,C 90.000,E1 200.972} C_DIS
LIN {X -0.013,Y -138.981,Z 1083.101,A 0.000,B 0.000,C 90.000,E1 198.181} C_DIS
LIN {X -0.052,Y -138.333,Z 1083.054,A 0.000,B 0.000,C 90.000,E1 189.792} C_DIS
LIN {X -0.028,Y -139.427,Z 1083.008,A 0.000,B 0.000,C 90.000,E1 181.375} C_DIS
LIN {X 0.026,Y -141.353,Z 1082.971,A 0.000,B 0.000,C 90.000,E1 174.837} C_DIS
LIN {X 0.002,Y -142.707,Z 1082.956,A 0.000,B 0.000,C 90.000,E1 172.064} C_DIS
LIN {X -0.039,Y -145.081,Z 1082.930,A 0.000,B 0.000,C 90.000,E1 167.465} C_DIS
LIN {X -0.043,Y -147.706,Z 1082.910,A 0.000,B 0.000,C 90.000,E1 163.795} C_DIS
LIN {X 0.040,Y -150.359,Z 1082.890,A 0.000,B 0.000,C 90.000,E1 160.115} C_DIS
LIN {X 0.059,Y -153.784,Z 1082.870,A 0.000,B 0.000,C 90.000,E1 156.485} C_DIS
LIN {X -0.020,Y -157.197,Z 1082.849,A 0.000,B 0.000,C 90.000,E1 152.922} C_DIS
LIN {X 0.061,Y -161.357,Z 1082.830,A 0.000,B 0.000,C 90.000,E1 149.331} C_DIS
LIN {X 0.073,Y -165.560,Z 1082.810,A 0.000,B 0.000,C 90.000,E1 145.801} C_DIS
LIN {X -0.044,Y -170.476,Z 1082.791,A 0.000,B 0.000,C 90.000,E1 142.351} C_DIS
LIN {X 0.106,Y -175.358,Z 1082.772,A 0.000,B 0.000,C 90.000,E1 138.852} C_DIS
LIN {X -0.031,Y -180.982,Z 1082.753,A 0.000,B 0.000,C 90.000,E1 135.486} C_DIS
LIN {X -0.044,Y -186.407,Z 1082.734,A 0.000,B 0.000,C 90.000,E1 132.123} C_DIS
LIN {X -0.105,Y -191.035,Z 1082.720,A 0.000,B 0.000,C 90.000,E1 129.644} C_DIS
LIN {X 0.088,Y -196.818,Z 1082.702,A 0.000,B 0.000,C 90.000,E1 126.297} C_DIS
LIN {X 0.002,Y -199.482,Z 1082.694,A 0.000,B 0.000,C 90.000,E1 124.978} C_DIS
LIN {X -0.045,Y -306.684,Z 1082.694,A 0.000,B 0.000,C 90.000,E1 124.978} C_DIS
LIN {X 0.038,Y -307.974,Z 1082.694,A 0.000,B 0.000,C 90.000,E1 124.945} C_DIS
LIN {X 0.009,Y -313.559,Z 1082.693,A 0.000,B 0.000,C 90.000,E1 124.692} C_DIS
LIN {X 0.002,Y -316.643,Z 1082.691,A 0.000,B 0.000,C 90.000,E1 124.405} C_DIS
LIN {X 0.055,Y -320.309,Z 1082.688,A 0.000,B 0.000,C 90.000,E1 123.865} C_DIS
LIN {X -0.142,Y -321.865,Z 1082.686,A 0.000,B 0.000,C 90.000,E1 123.579} C_DIS
LIN {X 0.021,Y -333.510,Z 1082.669,A 0.000,B 0.000,C 90.000,E1 120.384} C_DIS
LIN {X 0.025,Y -345.283,Z 1082.653,A 0.000,B 0.000,C 90.000,E1 117.590} C_DIS
LIN {X 0.070,Y -358.501,Z 1082.638,A 0.000,B 0.000,C 90.000,E1 114.847} C_DIS
LIN {X 0.101,Y -371.565,Z 1082.625,A 0.000,B 0.000,C 90.000,E1 112.461} C_DIS
LIN {X 0.172,Y -385.959,Z 1082.612,A 0.000,B 0.000,C 90.000,E1 110.120} C_DIS
LIN {X -0.037,Y -401.783,Z 1082.599,A 0.000,B 0.000,C 90.000,E1 107.873} C_DIS
LIN {X -0.116,Y -419.152,Z 1082.587,A 0.000,B 0.000,C 90.000,E1 105.662} C_DIS
LIN {X 0.035,Y -438.170,Z 1082.575,A 0.000,B 0.000,C 90.000,E1 103.480} C_DIS
LIN {X -0.185,Y -458.238,Z 1082.564,A 0.000,B 0.000,C 90.000,E1 101.478} C_DIS
LIN {X 0.120,Y -468.386,Z 1082.558,A 0.000,B 0.000,C 90.000,E1 100.489} C_DIS
LIN {X 0.144,Y -470.300,Z 1082.557,A 0.000,B 0.000,C 90.000,E1 100.254} C_DIS
LIN {X -0.004,Y -471.877,Z 1082.556,A 0.000,B 0.000,C 90.000,E1 100.018} C_DIS
LIN {X -0.154,Y -473.059,Z 1082.554,A 0.000,B 0.000,C 90.000,E1 99.782} C_DIS
LIN {X -0.048,Y -474.492,Z 1082.551,A 0.000,B 0.000,C 90.000,E1 99.265} C_DIS
LIN {X 0.069,Y -474.894,Z 1082.549,A 0.000,B 0.000,C 90.000,E1 98.746} C_DIS
LIN {X -0.203,Y -474.332,Z 1082.546,A 0.000,B 0.000,C 90.000,E1 98.276} C_DIS
LIN {X -0.076,Y -472.723,Z 1082.543,A 0.000,B 0.000,C 90.000,E1 97.757} C_DIS
LIN {X 0.191,Y -471.438,Z 1082.542,A 0.000,B 0.000,C 90.000,E1 97.473} C_DIS
LIN {X -0.142,Y -459.015,Z 1082.532,A 0.000,B 0.000,C 90.000,E1 95.739} C_DIS
LIN {X 0.141,Y -449.958,Z 1082.525,A 0.000,B 0.000,C 90.000,E1 94.416} C_DIS
LIN {X 0.197,Y -437.874,Z 1082.515,A 0.000,B 0.000,C 90.000,E1 92.579} C_DIS
LIN {X -0.170,Y -423.420,Z 1082.501,A 0.000,B 0.000,C 90.000,E1 90.229} C_DIS
LIN {X 0.101,Y -406.898,Z 1082.484,A 0.000,B 0.000,C 90.000,E1 87.192} C_DIS
LIN {X 0.082,Y -397.919,Z 1082.475,A 0.000,B 0.000,C 90.000,E1 85.527} C_DIS
LIN {X -0.058,Y -388.690,Z 1082.466,A 0.000,B 0.000,C 90.000,E1 83.856} C_DIS
LIN {X 0.020,Y -379.474,Z 1082.456,A 0.000,B 0.000,C 90.000,E1 82.129} C_DIS
LIN {X 0.030,Y -369.997,Z 1082.447,A 0.000,B 0.000,C 90.000,E1 80.387} C_DIS
LIN {X -0.059,Y -360.210,Z 1082.437,A 0.000,B 0.000,C 90.000,E1 78.634} C_DIS
LIN {X 0.024,Y -350.259,Z 1082.427,A 0.000,B 0.000,C 90.000,E1 76.825} C_DIS
LIN {X -0.025,Y -336.979,Z 1082.413,A 0.000,B 0.000,C 90.000,E1 74.393} C_DIS
LIN {X -0.032,Y -322.575,Z 1082.398,A 0.000,B 0.000,C 90.000,E1 71.583} C_DIS
LIN {X 0.106,Y -306.132,Z 1082.378,A 0.000,B 0.000,C 90.000,E1 68.028} C_DIS
LIN {X 0.037,Y -296.129,Z 1082.365,A 0.000,B 0.000,C 90.000,E1 65.741} C_DIS
LIN {X 0.117,Y -286.328,Z 1082.352,A 0.000,B 0.000,C 90.000,E1 63.384} C_DIS
LIN {X 0.058,Y -275.349,Z 1082.337,A 0.000,B 0.000,C 90.000,E1 60.667} C_DIS
LIN {X -0.096,Y -264.698,Z 1082.322,A 0.000,B 0.000,C 90.000,E1 57.916} C_DIS
LIN {X -0.006,Y -254.405,Z 1082.306,A 0.000,B 0.000,C 90.000,E1 55.055} C_DIS
LIN {X 0.043,Y -243.398,Z 1082.288,A 0.000,B 0.000,C 90.000,E1 51.778} C_DIS
LIN {X 0.022,Y -233.090,Z 1082.269,A 0.000,B 0.000,C 90.000,E1 48.447} C_DIS
LIN {X 0.105,Y -224.525,Z 1082.252,A 0.000,B 0.000,C 90.000,E1 45.405} C_DIS
LIN {X -0.020,Y -216.357,Z 1082.235,A 0.000,B 0.000,C 90.000,E1 42.366} C_DIS
LIN {X -0.016,Y -208.566,Z 1082.218,A 0.000,B 0.000,C 90.000,E1 39.241} C_DIS
LIN {X -0.108,Y -201.306,Z 1082.200,A 0.000,B 0.000,C 90.000,E1 36.091} C_DIS
LIN {X 0.005,Y -194.651,Z 1082.182,A 0.000,B 0.000,C 90.000,E1 32.832} C_DIS
LIN {X 0.067,Y -188.644,Z 1082.164,A 0.000,B 0.000,C 90.000,E1 29.539} C_DIS
LIN {X 0.030,Y -183.434,Z 1082.146,A 0.000,B 0.000,C 90.000,E1 26.232} C_DIS
LIN {X -0.041,Y -178.924,Z 1082.127,A 0.000,B 0.000,C 90.000,E1 22.898} C_DIS
LIN {X -0.031,Y -175.071,Z 1082.108,A 0.000,B 0.000,C 90.000,E1 19.504} C_DIS
LIN {X 0.070,Y -171.248,Z 1082.084,A 0.000,B 0.000,C 90.000,E1 15.190} C_DIS
LIN {X 0.036,Y -168.051,Z 1082.056,A 0.000,B 0.000,C 90.000,E1 10.018} C_DIS
LIN {X -0.077,Y -165.973,Z 1082.017,A 0.000,B 0.000,C 90.000,E1 3.094} C_DIS
LIN {X 0.050,Y -167.420,Z 1081.959,A 0.000,B 0.000,C 90.000,E1 352.534} C_DIS
LIN {X -0.071,Y -169.678,Z 1081.934,A 0.000,B 0.000,C 90.000,E1 348.229} C_DIS
LIN {X 0.059,Y -173.003,Z 1081.911,A 0.000,B 0.000,C 90.000,E1 343.866} C_DIS
LIN {X 0.092,Y -177.422,Z 1081.887,A 0.000,B 0.000,C 90.000,E1 339.571} C_DIS
LIN {X -0.074,Y -181.672,Z 1081.868,A 0.000,B 0.000,C 90.000,E1 336.230} C_DIS
LIN {X -0.086,Y -186.626,Z 1081.849,A 0.000,B 0.000,C 90.000,E1 332.871} C_DIS
LIN {X -0.051,Y -192.392,Z 1081.831,A 0.000,B 0.000,C 90.000,E1 329.537} C_DIS
LIN {X 0.100,Y -199.034,Z 1081.813,A 0.000,B 0.000,C 90.000,E1 326.215} C_DIS
LIN {X 0.031,Y -206.370,Z 1081.795,A 0.000,B 0.000,C 90.000,E1 323.004} C_DIS
LIN {X -0.065,Y -215.407,Z 1081.775,A 0.000,B 0.000,C 90.000,E1 319.461} C_DIS
LIN {X -0.091,Y -225.471,Z 1081.755,A 0.000,B 0.000,C 90.000,E1 315.972} C_DIS
LIN {X -0.110,Y -235.488,Z 1081.738,A 0.000,B 0.000,C 90.000,E1 312.933} C_DIS
LIN {X 0.009,Y -243.914,Z 1081.726,A 0.000,B 0.000,C 90.000,E1 310.663} C_DIS
LIN {X 0.024,Y -255.143,Z 1081.712,A 0.000,B 0.000,C 90.000,E1 308.096} C_DIS
LIN {X 0.084,Y -265.680,Z 1081.700,A 0.000,B 0.000,C 90.000,E1 305.931} C_DIS
LIN {X 0.006,Y -282.941,Z 1081.682,A 0.000,B 0.000,C 90.000,E1 302.801} C_DIS
LIN {X 0.074,Y -301.729,Z 1081.665,A 0.000,B 0.000,C 90.000,E1 299.745} C_DIS
LIN {X 0.067,Y -319.740,Z 1081.651,A 0.000,B 0.000,C 90.000,E1 297.129} C_DIS
LIN {X -0.208,Y -334.154,Z 1081.640,A 0.000,B 0.000,C 90.000,E1 295.283} C_DIS
LIN {X -0.058,Y -349.775,Z 1081.630,A 0.000,B 0.000,C 90.000,E1 293.439} C_DIS
LIN {X 0.040,Y -365.815,Z 1081.621,A 0.000,B 0.000,C 90.000,E1 291.770} C_DIS
LIN {X -0.159,Y -393.325,Z 1081.607,A 0.000,B 0.000,C 90.000,E1 289.322} C_DIS
LIN {X 0.051,Y -404.199,Z 1081.602,A 0.000,B 0.000,C 90.000,E1 288.362} C_DIS
LIN {X -0.151,Y -414.844,Z 1081.597,A 0.000,B 0.000,C 90.000,E1 287.457} C_DIS
LIN {X -0.136,Y -422.705,Z 1081.593,A 0.000,B 0.000,C 90.000,E1 286.732} C_DIS
LIN {X 0.075,Y -430.249,Z 1081.589,A 0.000,B 0.000,C 90.000,E1 285.969} C_DIS
LIN {X 0.116,Y -437.680,Z 1081.584,A 0.000,B 0.000,C 90.000,E1 285.190} C_DIS
LIN {X 0.004,Y -444.880,Z 1081.580,A 0.000,B 0.000,C 90.000,E1 284.411} C_DIS
LIN {X -0.189,Y -451.501,Z 1081.576,A 0.000,B 0.000,C 90.000,E1 283.647} C_DIS
LIN {X 0.126,Y -457.568,Z 1081.571,A 0.000,B 0.000,C 90.000,E1 282.827} C_DIS
LIN {X 0.048,Y -462.946,Z 1081.567,A 0.000,B 0.000,C 90.000,E1 282.063} C_DIS
LIN {X 0.176,Y -466.116,Z 1081.564,A 0.000,B 0.000,C 90.000,E1 281.535} C_DIS
LIN {X 0.086,Y -470.160,Z 1081.560,A 0.000,B 0.000,C 90.000,E1 280.782} C_DIS
LIN {X 0.115,Y -473.561,Z 1081.556,A 0.000,B 0.000,C 90.000,E1 280.018} C_DIS
LIN {X -0.244,Y -475.511,Z 1081.553,A 0.000,B 0.000,C 90.000,E1 279.557} C_DIS
LIN {X -0.049,Y -477.217,Z 1081.550,A 0.000,B 0.000,C 90.000,E1 279.029} C_DIS
LIN {X 0.083,Y -478.678,Z 1081.547,A 0.000,B 0.000,C 90.000,E1 278.511} C_DIS
LIN {X -0.248,Y -479.942,Z 1081.545,A 0.000,B 0.000,C 90.000,E1 278.049} C_DIS
LIN {X 0.129,Y -481.834,Z 1081.539,A 0.000,B 0.000,C 90.000,E1 277.004} C_DIS
LIN {X -0.183,Y -482.487,Z 1081.536,A 0.000,B 0.000,C 90.000,E1 276.543} C_DIS
LIN {X -0.063,Y -482.930,Z 1081.533,A 0.000,B 0.000,C 90.000,E1 276.030} C_DIS
LIN {X 0.116,Y -482.976,Z 1081.531,A 0.000,B 0.000,C 90.000,E1 275.511} C_DIS
LIN {X -0.184,Y -482.649,Z 1081.528,A 0.000,B 0.000,C 90.000,E1 275.049} C_DIS
LIN {X -0.005,Y -481.866,Z 1081.525,A 0.000,B 0.000,C 90.000,E1 274.531} C_DIS
LIN {X 0.168,Y -480.605,Z 1081.522,A 0.000,B 0.000,C 90.000,E1 274.012} C_DIS
LIN {X -0.174,Y -478.734,Z 1081.520,A 0.000,B 0.000,C 90.000,E1 273.555} C_DIS
LIN {X -0.015,Y -476.239,Z 1081.517,A 0.000,B 0.000,C 90.000,E1 273.037} C_DIS
LIN {X 0.099,Y -472.946,Z 1081.514,A 0.000,B 0.000,C 90.000,E1 272.522} C_DIS
LIN {X 0.199,Y -468.770,Z 1081.511,A 0.000,B 0.000,C 90.000,E1 272.007} C_DIS
LIN {X -0.174,Y -463.563,Z 1081.508,A 0.000,B 0.000,C 90.000,E1 271.547} C_DIS
LIN {X 0.168,Y -457.613,Z 1081.506,A 0.000,B 0.000,C 90.000,E1 271.031} C_DIS
LIN {X -0.018,Y -451.025,Z 1081.504,A 0.000,B 0.000,C 90.000,E1 270.630} C_DIS
LIN {X -0.096,Y -444.075,Z 1081.501,A 0.000,B 0.000,C 90.000,E1 270.286} C_DIS
LIN {X -0.095,Y -436.830,Z 1081.500,A 0.000,B 0.000,C 90.000,E1 270.000} C_DIS
LIN {X -0.086,Y -428.924,Z 1081.499,A 0.000,B 0.000,C 90.000,E1 269.771} C_DIS
LIN {X -0.069,Y -421.084,Z 1081.498,A 0.000,B 0.000,C 90.000,E1 269.599} C_DIS
LIN {X -0.165,Y -412.862,Z 1081.497,A 0.000,B 0.000,C 90.000,E1 269.484} C_DIS
LIN {X -0.043,Y -403.303,Z 1081.496,A 0.000,B 0.000,C 90.000,E1 269.370} C_DIS
LIN {X 0.037,Y -392.544,Z 1081.496,A 0.000,B 0.000,C 90.000,E1 269.312} C_DIS
LIN {X -0.011,Y -181.391,Z 1081.496,A 0.000,B 0.000,C 90.000,E1 269.312} C_DIS
LIN {X 0.078,Y -180.786,Z 1081.471,A 0.000,B 0.000,C 90.000,E1 264.723} C_DIS
LIN {X -0.028,Y -178.883,Z 1081.443,A 0.000,B 0.000,C 90.000,E1 259.690} C_DIS
LIN {X 0.048,Y -175.926,Z 1081.414,A 0.000,B 0.000,C 90.000,E1 254.574} C_DIS
LIN {X -0.007,Y -175.366,Z 1081.410,A 0.000,B 0.000,C 90.000,E1 253.740} C_DIS
LIN {X 0.052,Y -172.143,Z 1081.386,A 0.000,B 0.000,C 90.000,E1 249.444} C_DIS
LIN {X 0.029,Y -171.607,Z 1081.381,A 0.000,B 0.000,C 90.000,E1 248.592} C_DIS
LIN {X 0.017,Y -167.831,Z 1081.357,A 0.000,B 0.000,C 90.000,E1 244.280} C_DIS
LIN {X 0.034,Y -166.556,Z 1081.348,A 0.000,B 0.000,C 90.000,E1 242.538} C_DIS
LIN {X -0.055,Y -162.550,Z 1081.323,A 0.000,B 0.000,C 90.000,E1 238.201} C_DIS
LIN {X 0.005,Y -161.229,Z 1081.313,A 0.000,B 0.000,C 90.000,E1 236.421} C_DIS
LIN {X 0.040,Y -157.235,Z 1081.289,A 0.000,B 0.000,C 90.000,E1 231.984} C_DIS
LIN {X 0.062,Y -155.959,Z 1081.279,A 0.000,B 0.000,C 90.000,E1 230.194} C_DIS
LIN {X 0.021,Y -152.213,Z 1081.254,A 0.000,B 0.000,C 90.000,E1 225.729} C_DIS
LIN {X 0.042,Y -150.457,Z 1081.239,A 0.000,B 0.000,C 90.000,E1 223.014} C_DIS
LIN {X 0.068,Y -147.182,Z 1081.214,A 0.000,B 0.000,C 90.000,E1 218.463} C_DIS
LIN {X 0.034,Y -145.200,Z 1081.193,A 0.000,B 0.000,C 90.000,E1 214.818} C_DIS
LIN {X -0.056,Y -142.338,Z 1081.163,A 0.000,B 0.000,C 90.000,E1 209.333} C_DIS
LIN {X -0.002,Y -141.726,Z 1081.153,A 0.000,B 0.000,C 90.000,E1 207.462} C_DIS
LIN {X -0.020,Y -139.480,Z 1081.116,A 0.000,B 0.000,C 90.000,E1 200.972} C_DIS
